// TIA Portal V21 export
FUNCTION_BLOCK "FB603"   // FB603, LAD
TITLE = FB603
{ S7_Optimized_Access := 'FALSE' }
AUTHOR : PRECISE
FAMILY : PRECISE
// CIP
// stored: AutoNumber false, SetENOAutomatically false
   VAR_INPUT
      CycleEnable : Bool;
      CycleRunning : Bool;
      SecPulse : Bool;
      AlwaysTrue : Bool;
      CycleSelection : "CIP";
      ConductivitySuccessWhileRinse : Bool;
      ConductivitySuccessWhileDrain : Bool;
      ConductivitySuccessWhileTransfer : Bool;
   END_VAR
   VAR_OUTPUT
      Started : Bool;
      VentValve : Bool;
      PrintActualRep : Int;
   END_VAR
   VAR_IN_OUT
      Over : Bool;
      OverTemp : Bool;
      RepeatCycle : Bool;
      ActualRepetition : Int;
      CycleStart : "CipCycleStarted";
      CycleOver : "CipCycleOver";
      ConductivityStatus : Bool;
      TimeSaveModeRep : Int;
      StartFillingToSaveTime : Bool;
      Reset : Bool;
      RecirculationPopupTemp : Bool;
      RecirculationPopupTempAck : Bool;
   END_VAR
   VAR
      Re : Array[0..30] of Bool;
   END_VAR
   VAR_TEMP   // added for the SCL form of the ladder/FBD networks
      _w1 : Bool;
      _w2 : Bool;
      _w3 : Bool;
      _w4 : Bool;
      _w5 : Bool;
      _w6 : Bool;
      _w7 : Bool;
      _w8 : Bool;
      _w9 : Bool;
      _w10 : Bool;
      _w11 : Bool;
      _w12 : Bool;
   END_VAR
BEGIN

REGION Network 1
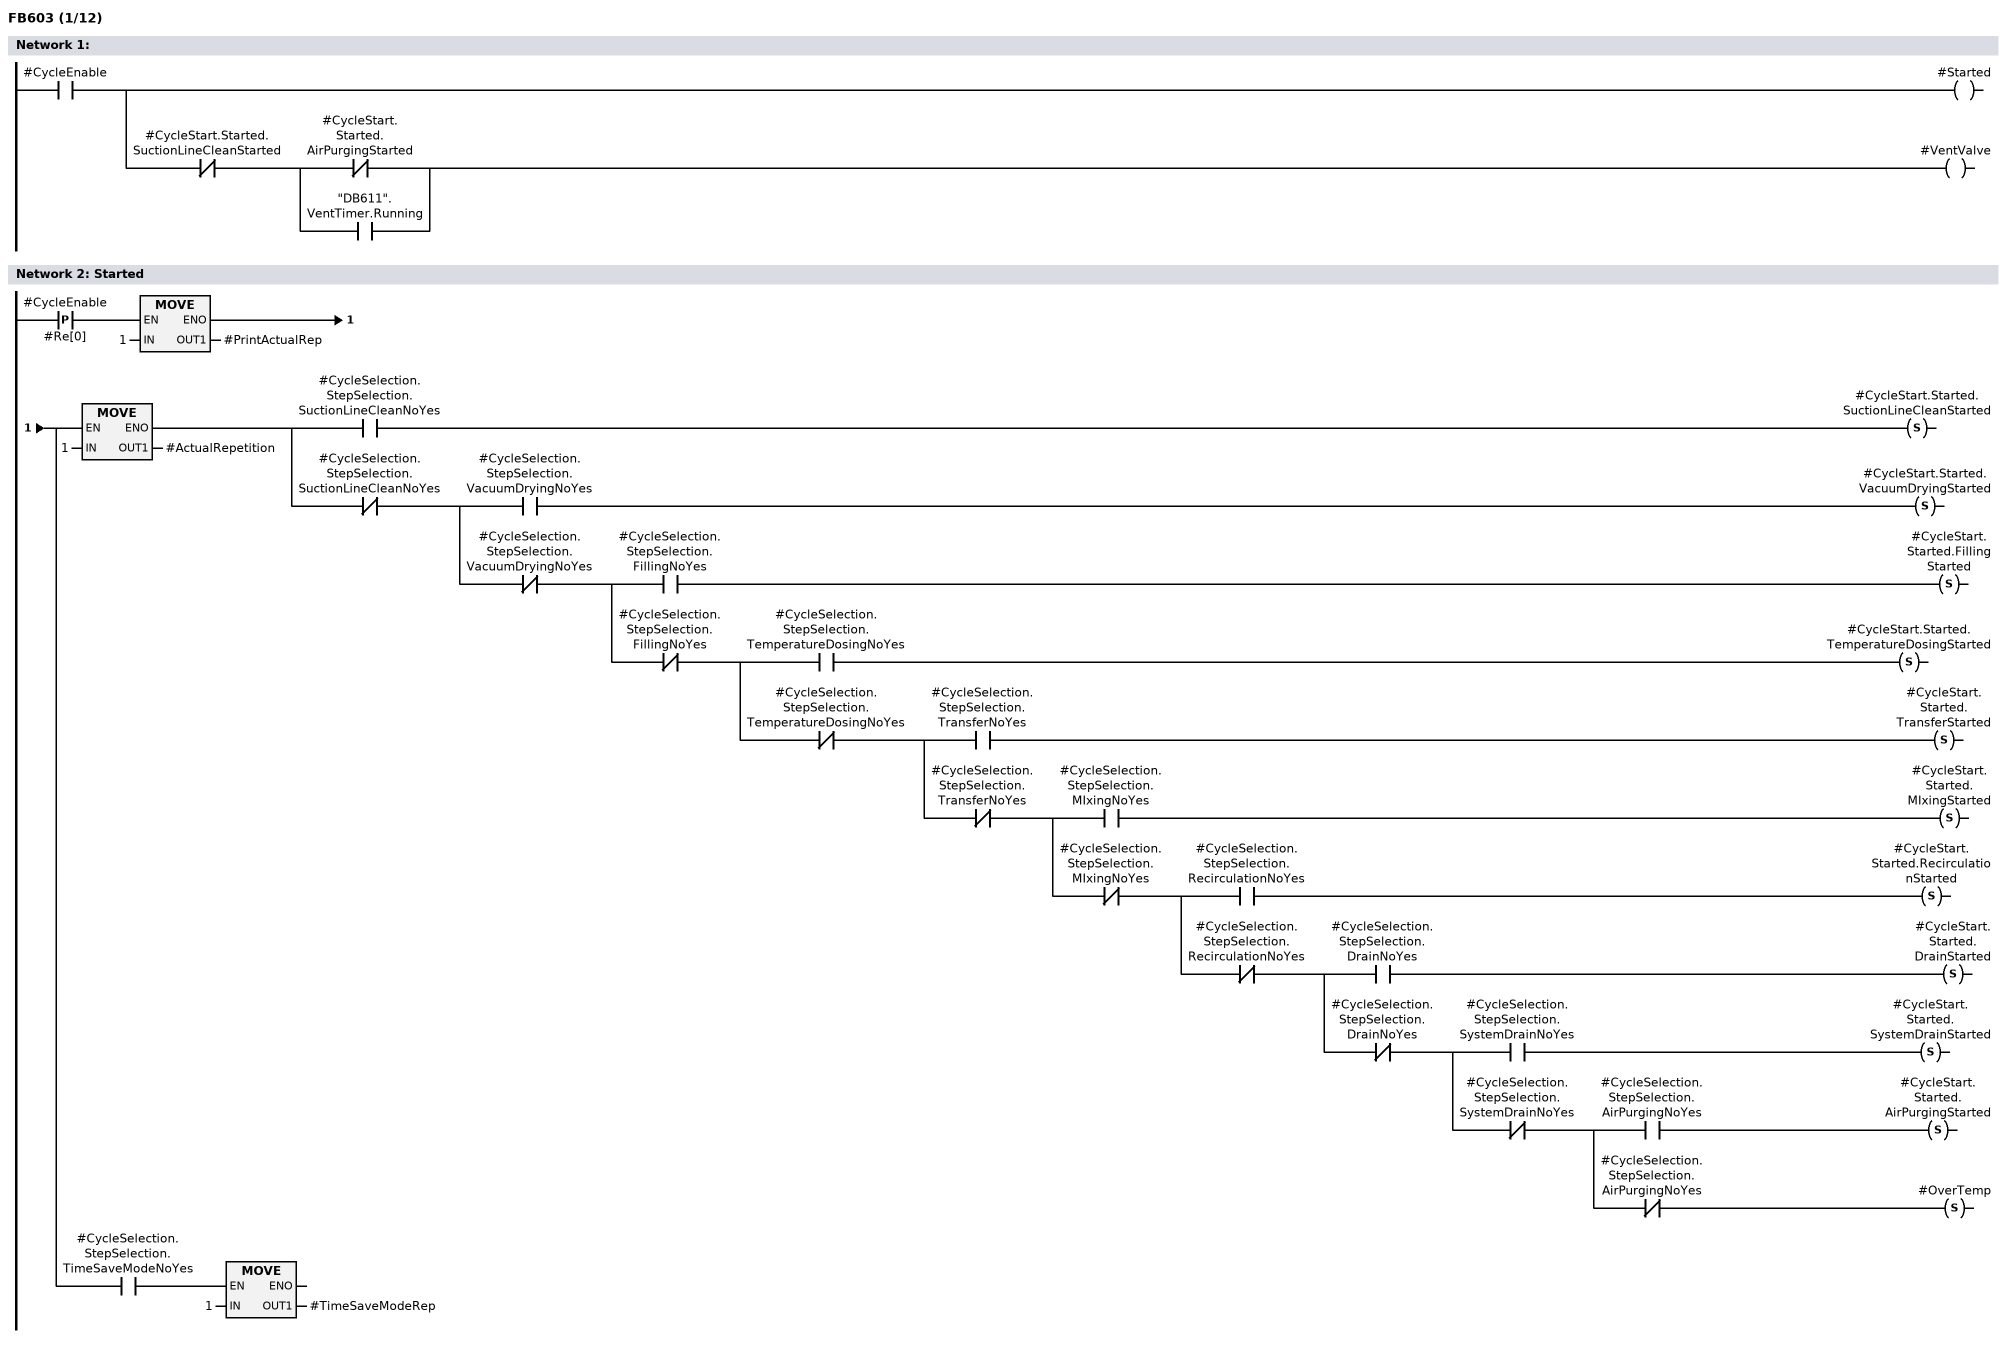
   RUNG wire#powerrail
      Contact( #CycleEnable )
      wire#w1
      Coil( #Started )
   END_RUNG
   RUNG wire#w1
      I_Contact( #CycleStart.Started.SuctionLineCleanStarted )
      wire#w2
      I_Contact( #CycleStart.Started.AirPurgingStarted )
      wire#w3
      Coil( #VentValve )
   END_RUNG
   RUNG wire#w2
      Contact( "DB611".VentTimer.Running )
   END_RUNG wire#w3
   // the same network as SCL:
   #Started := #CycleEnable;
   #VentValve := #CycleEnable AND NOT #CycleStart.Started.SuctionLineCleanStarted AND (NOT #CycleStart.Started.AirPurgingStarted OR "DB611".VentTimer.Running);
END_REGION

REGION Network 2: Started
   RUNG wire#powerrail
      P_Contact(operand := #CycleEnable, bit := #Re[0])
      Move(in := 1, out1 => #PrintActualRep)
      wire#w1
      Move(in := 1, out1 => #ActualRepetition)
      wire#w2
      Contact( #CycleSelection.StepSelection.SuctionLineCleanNoYes )
      S_Coil( #CycleStart.Started.SuctionLineCleanStarted )
   END_RUNG
   RUNG wire#w2
      I_Contact( #CycleSelection.StepSelection.SuctionLineCleanNoYes )
      wire#w3
      Contact( #CycleSelection.StepSelection.VacuumDryingNoYes )
      S_Coil( #CycleStart.Started.VacuumDryingStarted )
   END_RUNG
   RUNG wire#w3
      I_Contact( #CycleSelection.StepSelection.VacuumDryingNoYes )
      wire#w4
      Contact( #CycleSelection.StepSelection.FillingNoYes )
      S_Coil( #CycleStart.Started.FillingStarted )
   END_RUNG
   RUNG wire#w4
      I_Contact( #CycleSelection.StepSelection.FillingNoYes )
      wire#w5
      Contact( #CycleSelection.StepSelection.TemperatureDosingNoYes )
      S_Coil( #CycleStart.Started.TemperatureDosingStarted )
   END_RUNG
   RUNG wire#w5
      I_Contact( #CycleSelection.StepSelection.TemperatureDosingNoYes )
      wire#w6
      Contact( #CycleSelection.StepSelection.TransferNoYes )
      S_Coil( #CycleStart.Started.TransferStarted )
   END_RUNG
   RUNG wire#w6
      I_Contact( #CycleSelection.StepSelection.TransferNoYes )
      wire#w7
      Contact( #CycleSelection.StepSelection.MIxingNoYes )
      S_Coil( #CycleStart.Started.MIxingStarted )
   END_RUNG
   RUNG wire#w7
      I_Contact( #CycleSelection.StepSelection.MIxingNoYes )
      wire#w8
      Contact( #CycleSelection.StepSelection.RecirculationNoYes )
      S_Coil( #CycleStart.Started.RecirculationStarted )
   END_RUNG
   RUNG wire#w8
      I_Contact( #CycleSelection.StepSelection.RecirculationNoYes )
      wire#w9
      Contact( #CycleSelection.StepSelection.DrainNoYes )
      S_Coil( #CycleStart.Started.DrainStarted )
   END_RUNG
   RUNG wire#w9
      I_Contact( #CycleSelection.StepSelection.DrainNoYes )
      wire#w10
      Contact( #CycleSelection.StepSelection.SystemDrainNoYes )
      S_Coil( #CycleStart.Started.SystemDrainStarted )
   END_RUNG
   RUNG wire#w10
      I_Contact( #CycleSelection.StepSelection.SystemDrainNoYes )
      wire#w11
      Contact( #CycleSelection.StepSelection.AirPurgingNoYes )
      S_Coil( #CycleStart.Started.AirPurgingStarted )
   END_RUNG
   RUNG wire#w11
      I_Contact( #CycleSelection.StepSelection.AirPurgingNoYes )
      S_Coil( #OverTemp )
   END_RUNG
   RUNG wire#w1
      Contact( #CycleSelection.StepSelection.TimeSaveModeNoYes )
      Move(in := 1, out1 => #TimeSaveModeRep)
   END_RUNG
   // the same network as SCL:
   #_w1 := #CycleEnable AND NOT #Re[0];   // rising edge of #CycleEnable
   #Re[0] := #CycleEnable;
   IF #_w1 THEN
       #PrintActualRep := 1;
       #ActualRepetition := 1;
   END_IF;
   IF #_w1 AND #CycleSelection.StepSelection.SuctionLineCleanNoYes THEN
       #CycleStart.Started.SuctionLineCleanStarted := TRUE;
   END_IF;
   #_w2 := #_w1 AND NOT #CycleSelection.StepSelection.SuctionLineCleanNoYes;
   IF #_w2 AND #CycleSelection.StepSelection.VacuumDryingNoYes THEN
       #CycleStart.Started.VacuumDryingStarted := TRUE;
   END_IF;
   #_w3 := #_w2 AND NOT #CycleSelection.StepSelection.VacuumDryingNoYes;
   IF #_w3 AND #CycleSelection.StepSelection.FillingNoYes THEN
       #CycleStart.Started.FillingStarted := TRUE;
   END_IF;
   #_w4 := #_w3 AND NOT #CycleSelection.StepSelection.FillingNoYes;
   IF #_w4 AND #CycleSelection.StepSelection.TemperatureDosingNoYes THEN
       #CycleStart.Started.TemperatureDosingStarted := TRUE;
   END_IF;
   #_w5 := #_w4 AND NOT #CycleSelection.StepSelection.TemperatureDosingNoYes;
   IF #_w5 AND #CycleSelection.StepSelection.TransferNoYes THEN
       #CycleStart.Started.TransferStarted := TRUE;
   END_IF;
   #_w6 := #_w5 AND NOT #CycleSelection.StepSelection.TransferNoYes;
   IF #_w6 AND #CycleSelection.StepSelection.MIxingNoYes THEN
       #CycleStart.Started.MIxingStarted := TRUE;
   END_IF;
   #_w7 := #_w6 AND NOT #CycleSelection.StepSelection.MIxingNoYes;
   IF #_w7 AND #CycleSelection.StepSelection.RecirculationNoYes THEN
       #CycleStart.Started.RecirculationStarted := TRUE;
   END_IF;
   #_w8 := #_w7 AND NOT #CycleSelection.StepSelection.RecirculationNoYes;
   IF #_w8 AND #CycleSelection.StepSelection.DrainNoYes THEN
       #CycleStart.Started.DrainStarted := TRUE;
   END_IF;
   #_w9 := #_w8 AND NOT #CycleSelection.StepSelection.DrainNoYes;
   IF #_w9 AND #CycleSelection.StepSelection.SystemDrainNoYes THEN
       #CycleStart.Started.SystemDrainStarted := TRUE;
   END_IF;
   #_w10 := #_w9 AND NOT #CycleSelection.StepSelection.SystemDrainNoYes;
   IF #_w10 AND #CycleSelection.StepSelection.AirPurgingNoYes THEN
       #CycleStart.Started.AirPurgingStarted := TRUE;
   END_IF;
   IF #_w10 AND NOT #CycleSelection.StepSelection.AirPurgingNoYes THEN #OverTemp := TRUE; END_IF;
   IF #_w1 AND #CycleSelection.StepSelection.TimeSaveModeNoYes THEN #TimeSaveModeRep := 1; END_IF;
END_REGION

REGION Network 3: SuctionLineCleanOver
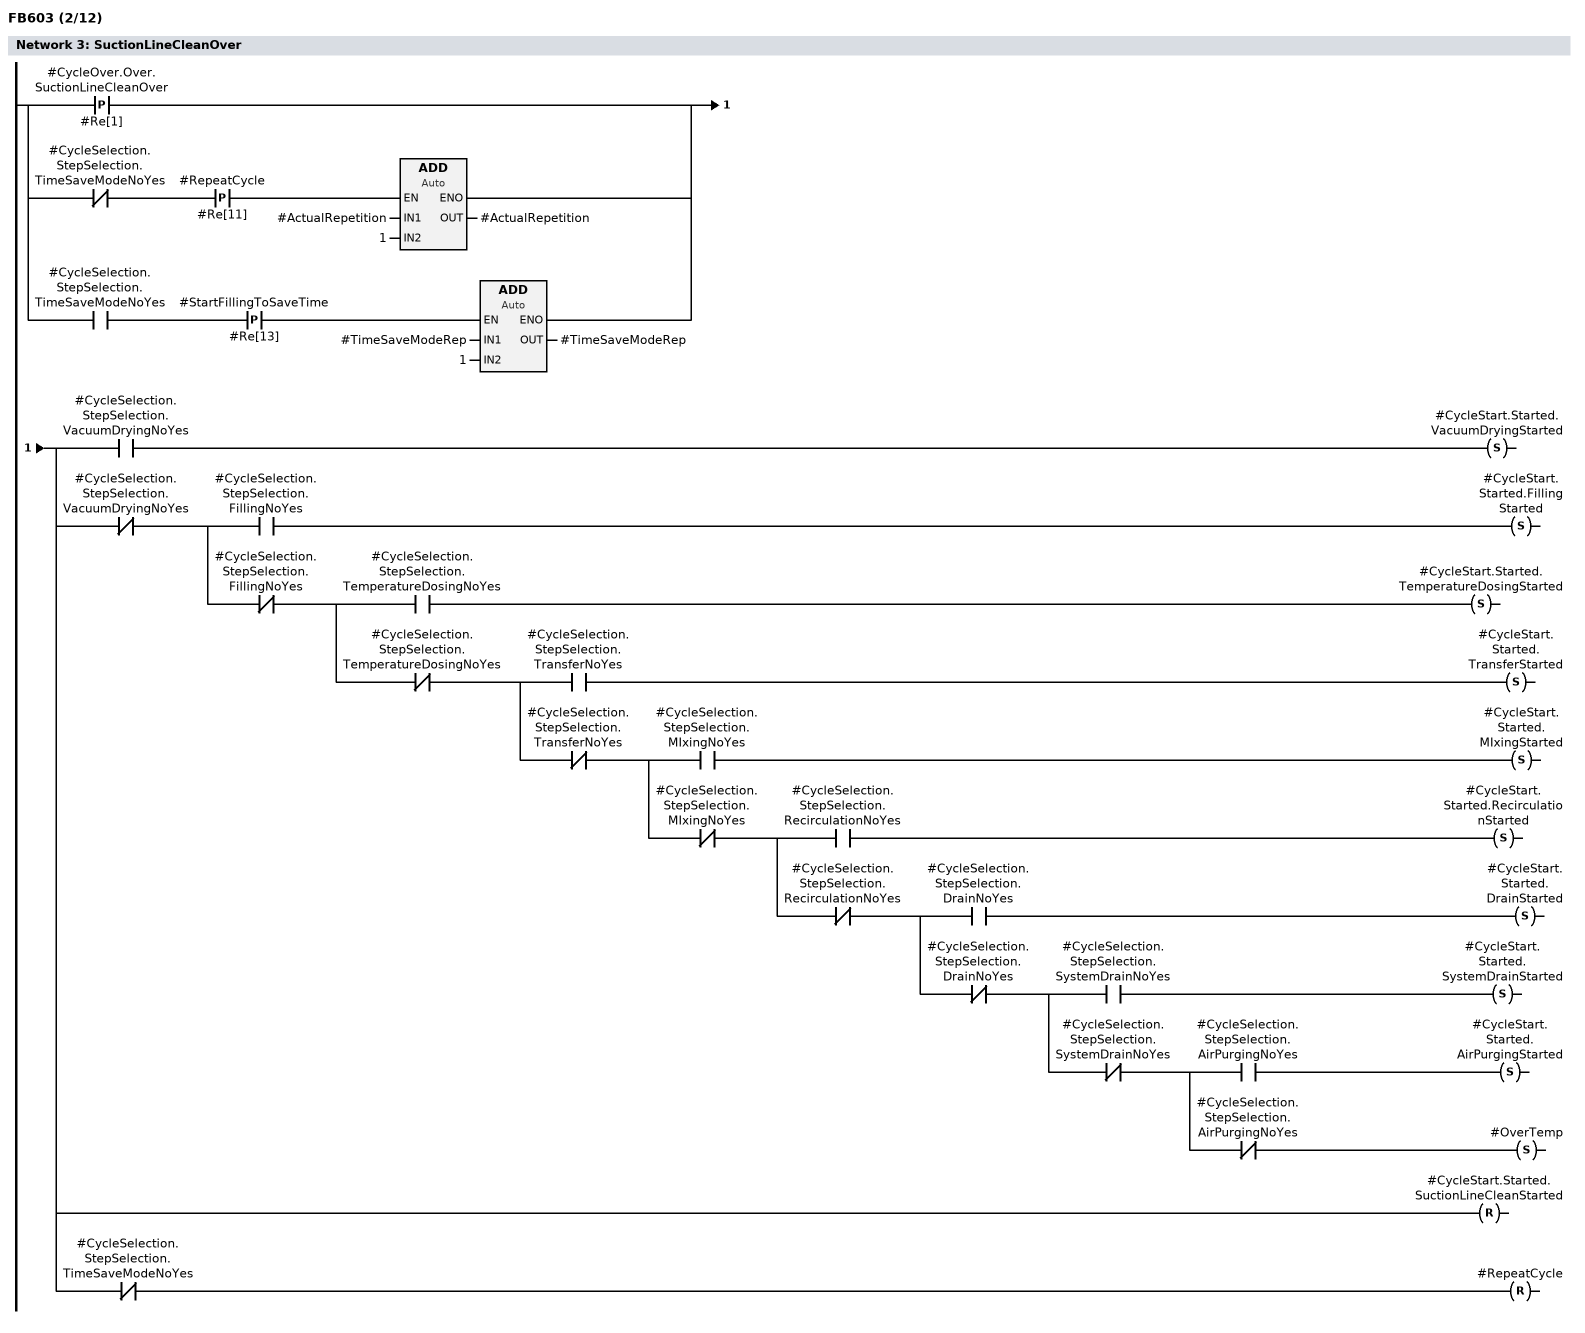
   RUNG wire#powerrail
      P_Contact(operand := #CycleOver.Over.SuctionLineCleanOver, bit := #Re[1])
      wire#w1
      Contact( #CycleSelection.StepSelection.VacuumDryingNoYes )
      S_Coil( #CycleStart.Started.VacuumDryingStarted )
   END_RUNG
   RUNG wire#powerrail
      I_Contact( #CycleSelection.StepSelection.TimeSaveModeNoYes )
      P_Contact(operand := #RepeatCycle, bit := #Re[11])
      Add(in1 := #ActualRepetition, in2 := 1, out => #ActualRepetition)
   END_RUNG wire#w1
   RUNG wire#powerrail
      Contact( #CycleSelection.StepSelection.TimeSaveModeNoYes )
      P_Contact(operand := #StartFillingToSaveTime, bit := #Re[13])
      Add(in1 := #TimeSaveModeRep, in2 := 1, out => #TimeSaveModeRep)
   END_RUNG wire#w1
   RUNG wire#w1
      I_Contact( #CycleSelection.StepSelection.VacuumDryingNoYes )
      wire#w2
      Contact( #CycleSelection.StepSelection.FillingNoYes )
      S_Coil( #CycleStart.Started.FillingStarted )
   END_RUNG
   RUNG wire#w2
      I_Contact( #CycleSelection.StepSelection.FillingNoYes )
      wire#w3
      Contact( #CycleSelection.StepSelection.TemperatureDosingNoYes )
      S_Coil( #CycleStart.Started.TemperatureDosingStarted )
   END_RUNG
   RUNG wire#w3
      I_Contact( #CycleSelection.StepSelection.TemperatureDosingNoYes )
      wire#w4
      Contact( #CycleSelection.StepSelection.TransferNoYes )
      S_Coil( #CycleStart.Started.TransferStarted )
   END_RUNG
   RUNG wire#w4
      I_Contact( #CycleSelection.StepSelection.TransferNoYes )
      wire#w5
      Contact( #CycleSelection.StepSelection.MIxingNoYes )
      S_Coil( #CycleStart.Started.MIxingStarted )
   END_RUNG
   RUNG wire#w5
      I_Contact( #CycleSelection.StepSelection.MIxingNoYes )
      wire#w6
      Contact( #CycleSelection.StepSelection.RecirculationNoYes )
      S_Coil( #CycleStart.Started.RecirculationStarted )
   END_RUNG
   RUNG wire#w6
      I_Contact( #CycleSelection.StepSelection.RecirculationNoYes )
      wire#w7
      Contact( #CycleSelection.StepSelection.DrainNoYes )
      S_Coil( #CycleStart.Started.DrainStarted )
   END_RUNG
   RUNG wire#w7
      I_Contact( #CycleSelection.StepSelection.DrainNoYes )
      wire#w8
      Contact( #CycleSelection.StepSelection.SystemDrainNoYes )
      S_Coil( #CycleStart.Started.SystemDrainStarted )
   END_RUNG
   RUNG wire#w8
      I_Contact( #CycleSelection.StepSelection.SystemDrainNoYes )
      wire#w9
      Contact( #CycleSelection.StepSelection.AirPurgingNoYes )
      S_Coil( #CycleStart.Started.AirPurgingStarted )
   END_RUNG
   RUNG wire#w9
      I_Contact( #CycleSelection.StepSelection.AirPurgingNoYes )
      S_Coil( #OverTemp )
   END_RUNG
   RUNG wire#w1
      R_Coil( #CycleStart.Started.SuctionLineCleanStarted )
   END_RUNG
   RUNG wire#w1
      I_Contact( #CycleSelection.StepSelection.TimeSaveModeNoYes )
      R_Coil( #RepeatCycle )
   END_RUNG
   // the same network as SCL:
   #_w1 := #CycleOver.Over.SuctionLineCleanOver AND NOT #Re[1];   // rising edge of #CycleOver.Over.SuctionLineCleanOver
   #Re[1] := #CycleOver.Over.SuctionLineCleanOver;
   #_w2 := NOT #CycleSelection.StepSelection.TimeSaveModeNoYes AND #RepeatCycle AND NOT #Re[11];   // rising edge of #RepeatCycle
   #Re[11] := #RepeatCycle;
   IF #_w2 THEN #ActualRepetition := #ActualRepetition + 1; END_IF;
   #_w3 := #CycleSelection.StepSelection.TimeSaveModeNoYes AND #StartFillingToSaveTime AND NOT #Re[13];   // rising edge of #StartFillingToSaveTime
   #Re[13] := #StartFillingToSaveTime;
   IF #_w3 THEN #TimeSaveModeRep := #TimeSaveModeRep + 1; END_IF;
   #_w4 := #_w1 OR #_w2 OR #_w3;
   IF #_w4 AND #CycleSelection.StepSelection.VacuumDryingNoYes THEN
       #CycleStart.Started.VacuumDryingStarted := TRUE;
   END_IF;
   #_w5 := #_w4 AND NOT #CycleSelection.StepSelection.VacuumDryingNoYes;
   IF #_w5 AND #CycleSelection.StepSelection.FillingNoYes THEN
       #CycleStart.Started.FillingStarted := TRUE;
   END_IF;
   #_w6 := #_w5 AND NOT #CycleSelection.StepSelection.FillingNoYes;
   IF #_w6 AND #CycleSelection.StepSelection.TemperatureDosingNoYes THEN
       #CycleStart.Started.TemperatureDosingStarted := TRUE;
   END_IF;
   #_w7 := #_w6 AND NOT #CycleSelection.StepSelection.TemperatureDosingNoYes;
   IF #_w7 AND #CycleSelection.StepSelection.TransferNoYes THEN
       #CycleStart.Started.TransferStarted := TRUE;
   END_IF;
   #_w8 := #_w7 AND NOT #CycleSelection.StepSelection.TransferNoYes;
   IF #_w8 AND #CycleSelection.StepSelection.MIxingNoYes THEN
       #CycleStart.Started.MIxingStarted := TRUE;
   END_IF;
   #_w9 := #_w8 AND NOT #CycleSelection.StepSelection.MIxingNoYes;
   IF #_w9 AND #CycleSelection.StepSelection.RecirculationNoYes THEN
       #CycleStart.Started.RecirculationStarted := TRUE;
   END_IF;
   #_w10 := #_w9 AND NOT #CycleSelection.StepSelection.RecirculationNoYes;
   IF #_w10 AND #CycleSelection.StepSelection.DrainNoYes THEN
       #CycleStart.Started.DrainStarted := TRUE;
   END_IF;
   #_w11 := #_w10 AND NOT #CycleSelection.StepSelection.DrainNoYes;
   IF #_w11 AND #CycleSelection.StepSelection.SystemDrainNoYes THEN
       #CycleStart.Started.SystemDrainStarted := TRUE;
   END_IF;
   #_w12 := #_w11 AND NOT #CycleSelection.StepSelection.SystemDrainNoYes;
   IF #_w12 AND #CycleSelection.StepSelection.AirPurgingNoYes THEN
       #CycleStart.Started.AirPurgingStarted := TRUE;
   END_IF;
   IF #_w12 AND NOT #CycleSelection.StepSelection.AirPurgingNoYes THEN #OverTemp := TRUE; END_IF;
   IF #_w4 THEN #CycleStart.Started.SuctionLineCleanStarted := FALSE; END_IF;
   IF #_w4 AND NOT #CycleSelection.StepSelection.TimeSaveModeNoYes THEN #RepeatCycle := FALSE; END_IF;
END_REGION

REGION Network 4: VacuumDryingOver
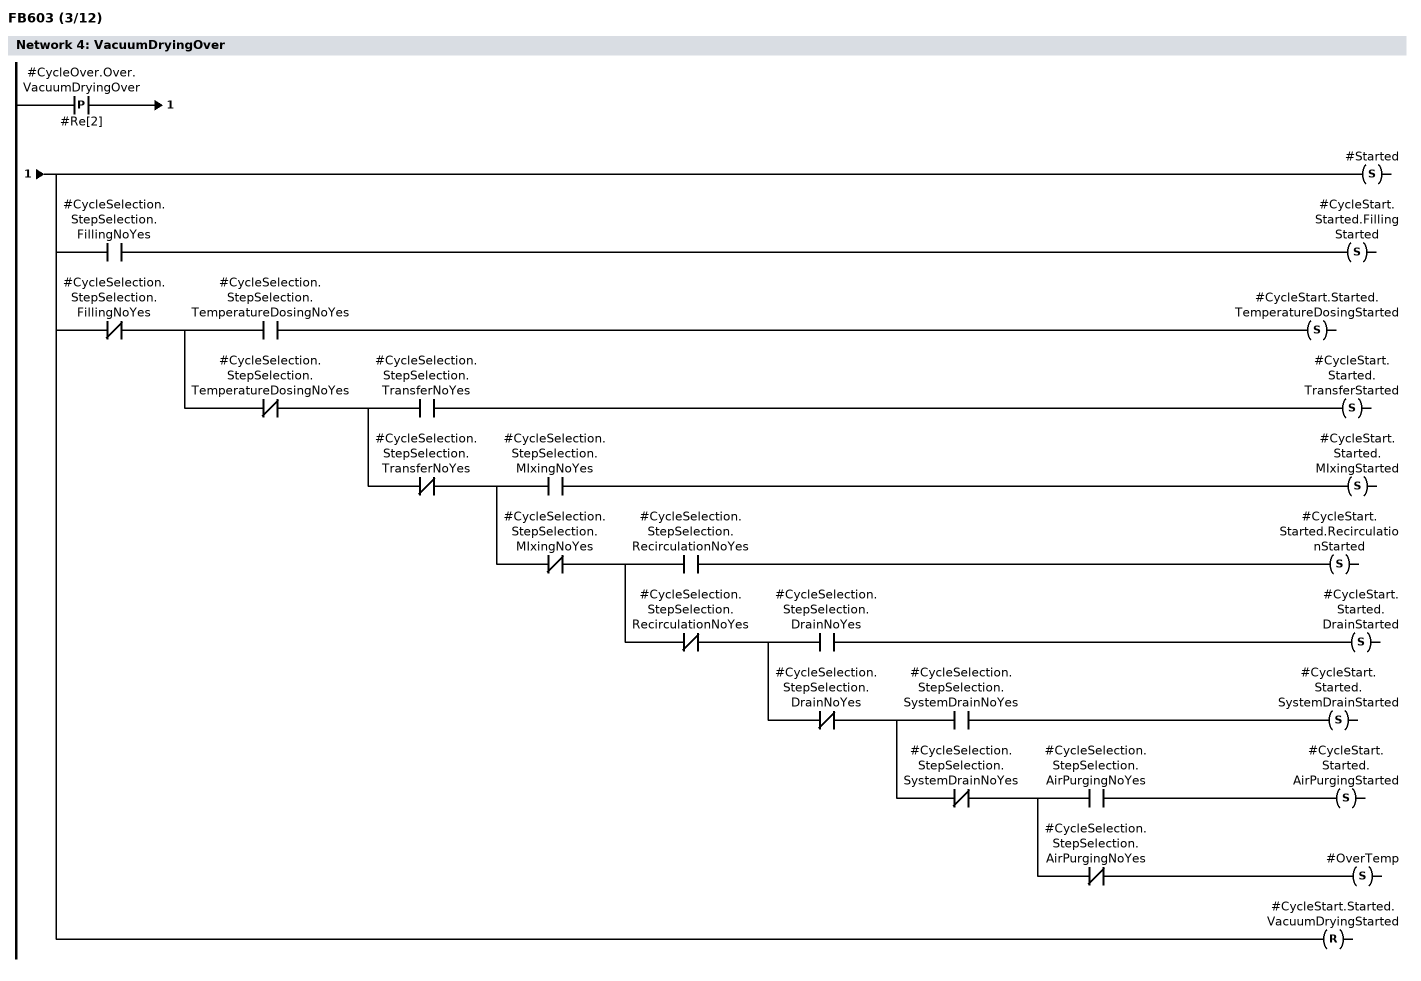
   RUNG wire#powerrail
      P_Contact(operand := #CycleOver.Over.VacuumDryingOver, bit := #Re[2])
      wire#w1
      S_Coil( #Started )
   END_RUNG
   RUNG wire#w1
      Contact( #CycleSelection.StepSelection.FillingNoYes )
      S_Coil( #CycleStart.Started.FillingStarted )
   END_RUNG
   RUNG wire#w1
      I_Contact( #CycleSelection.StepSelection.FillingNoYes )
      wire#w2
      Contact( #CycleSelection.StepSelection.TemperatureDosingNoYes )
      S_Coil( #CycleStart.Started.TemperatureDosingStarted )
   END_RUNG
   RUNG wire#w2
      I_Contact( #CycleSelection.StepSelection.TemperatureDosingNoYes )
      wire#w3
      Contact( #CycleSelection.StepSelection.TransferNoYes )
      S_Coil( #CycleStart.Started.TransferStarted )
   END_RUNG
   RUNG wire#w3
      I_Contact( #CycleSelection.StepSelection.TransferNoYes )
      wire#w4
      Contact( #CycleSelection.StepSelection.MIxingNoYes )
      S_Coil( #CycleStart.Started.MIxingStarted )
   END_RUNG
   RUNG wire#w4
      I_Contact( #CycleSelection.StepSelection.MIxingNoYes )
      wire#w5
      Contact( #CycleSelection.StepSelection.RecirculationNoYes )
      S_Coil( #CycleStart.Started.RecirculationStarted )
   END_RUNG
   RUNG wire#w5
      I_Contact( #CycleSelection.StepSelection.RecirculationNoYes )
      wire#w6
      Contact( #CycleSelection.StepSelection.DrainNoYes )
      S_Coil( #CycleStart.Started.DrainStarted )
   END_RUNG
   RUNG wire#w6
      I_Contact( #CycleSelection.StepSelection.DrainNoYes )
      wire#w7
      Contact( #CycleSelection.StepSelection.SystemDrainNoYes )
      S_Coil( #CycleStart.Started.SystemDrainStarted )
   END_RUNG
   RUNG wire#w7
      I_Contact( #CycleSelection.StepSelection.SystemDrainNoYes )
      wire#w8
      Contact( #CycleSelection.StepSelection.AirPurgingNoYes )
      S_Coil( #CycleStart.Started.AirPurgingStarted )
   END_RUNG
   RUNG wire#w8
      I_Contact( #CycleSelection.StepSelection.AirPurgingNoYes )
      S_Coil( #OverTemp )
   END_RUNG
   RUNG wire#w1
      R_Coil( #CycleStart.Started.VacuumDryingStarted )
   END_RUNG
   // the same network as SCL:
   #_w1 := #CycleOver.Over.VacuumDryingOver AND NOT #Re[2];   // rising edge of #CycleOver.Over.VacuumDryingOver
   #Re[2] := #CycleOver.Over.VacuumDryingOver;
   IF #_w1 THEN #Started := TRUE; END_IF;
   IF #_w1 AND #CycleSelection.StepSelection.FillingNoYes THEN
       #CycleStart.Started.FillingStarted := TRUE;
   END_IF;
   #_w2 := #_w1 AND NOT #CycleSelection.StepSelection.FillingNoYes;
   IF #_w2 AND #CycleSelection.StepSelection.TemperatureDosingNoYes THEN
       #CycleStart.Started.TemperatureDosingStarted := TRUE;
   END_IF;
   #_w3 := #_w2 AND NOT #CycleSelection.StepSelection.TemperatureDosingNoYes;
   IF #_w3 AND #CycleSelection.StepSelection.TransferNoYes THEN
       #CycleStart.Started.TransferStarted := TRUE;
   END_IF;
   #_w4 := #_w3 AND NOT #CycleSelection.StepSelection.TransferNoYes;
   IF #_w4 AND #CycleSelection.StepSelection.MIxingNoYes THEN
       #CycleStart.Started.MIxingStarted := TRUE;
   END_IF;
   #_w5 := #_w4 AND NOT #CycleSelection.StepSelection.MIxingNoYes;
   IF #_w5 AND #CycleSelection.StepSelection.RecirculationNoYes THEN
       #CycleStart.Started.RecirculationStarted := TRUE;
   END_IF;
   #_w6 := #_w5 AND NOT #CycleSelection.StepSelection.RecirculationNoYes;
   IF #_w6 AND #CycleSelection.StepSelection.DrainNoYes THEN
       #CycleStart.Started.DrainStarted := TRUE;
   END_IF;
   #_w7 := #_w6 AND NOT #CycleSelection.StepSelection.DrainNoYes;
   IF #_w7 AND #CycleSelection.StepSelection.SystemDrainNoYes THEN
       #CycleStart.Started.SystemDrainStarted := TRUE;
   END_IF;
   #_w8 := #_w7 AND NOT #CycleSelection.StepSelection.SystemDrainNoYes;
   IF #_w8 AND #CycleSelection.StepSelection.AirPurgingNoYes THEN
       #CycleStart.Started.AirPurgingStarted := TRUE;
   END_IF;
   IF #_w8 AND NOT #CycleSelection.StepSelection.AirPurgingNoYes THEN #OverTemp := TRUE; END_IF;
   IF #_w1 THEN #CycleStart.Started.VacuumDryingStarted := FALSE; END_IF;
END_REGION

REGION Network 5: FillOver
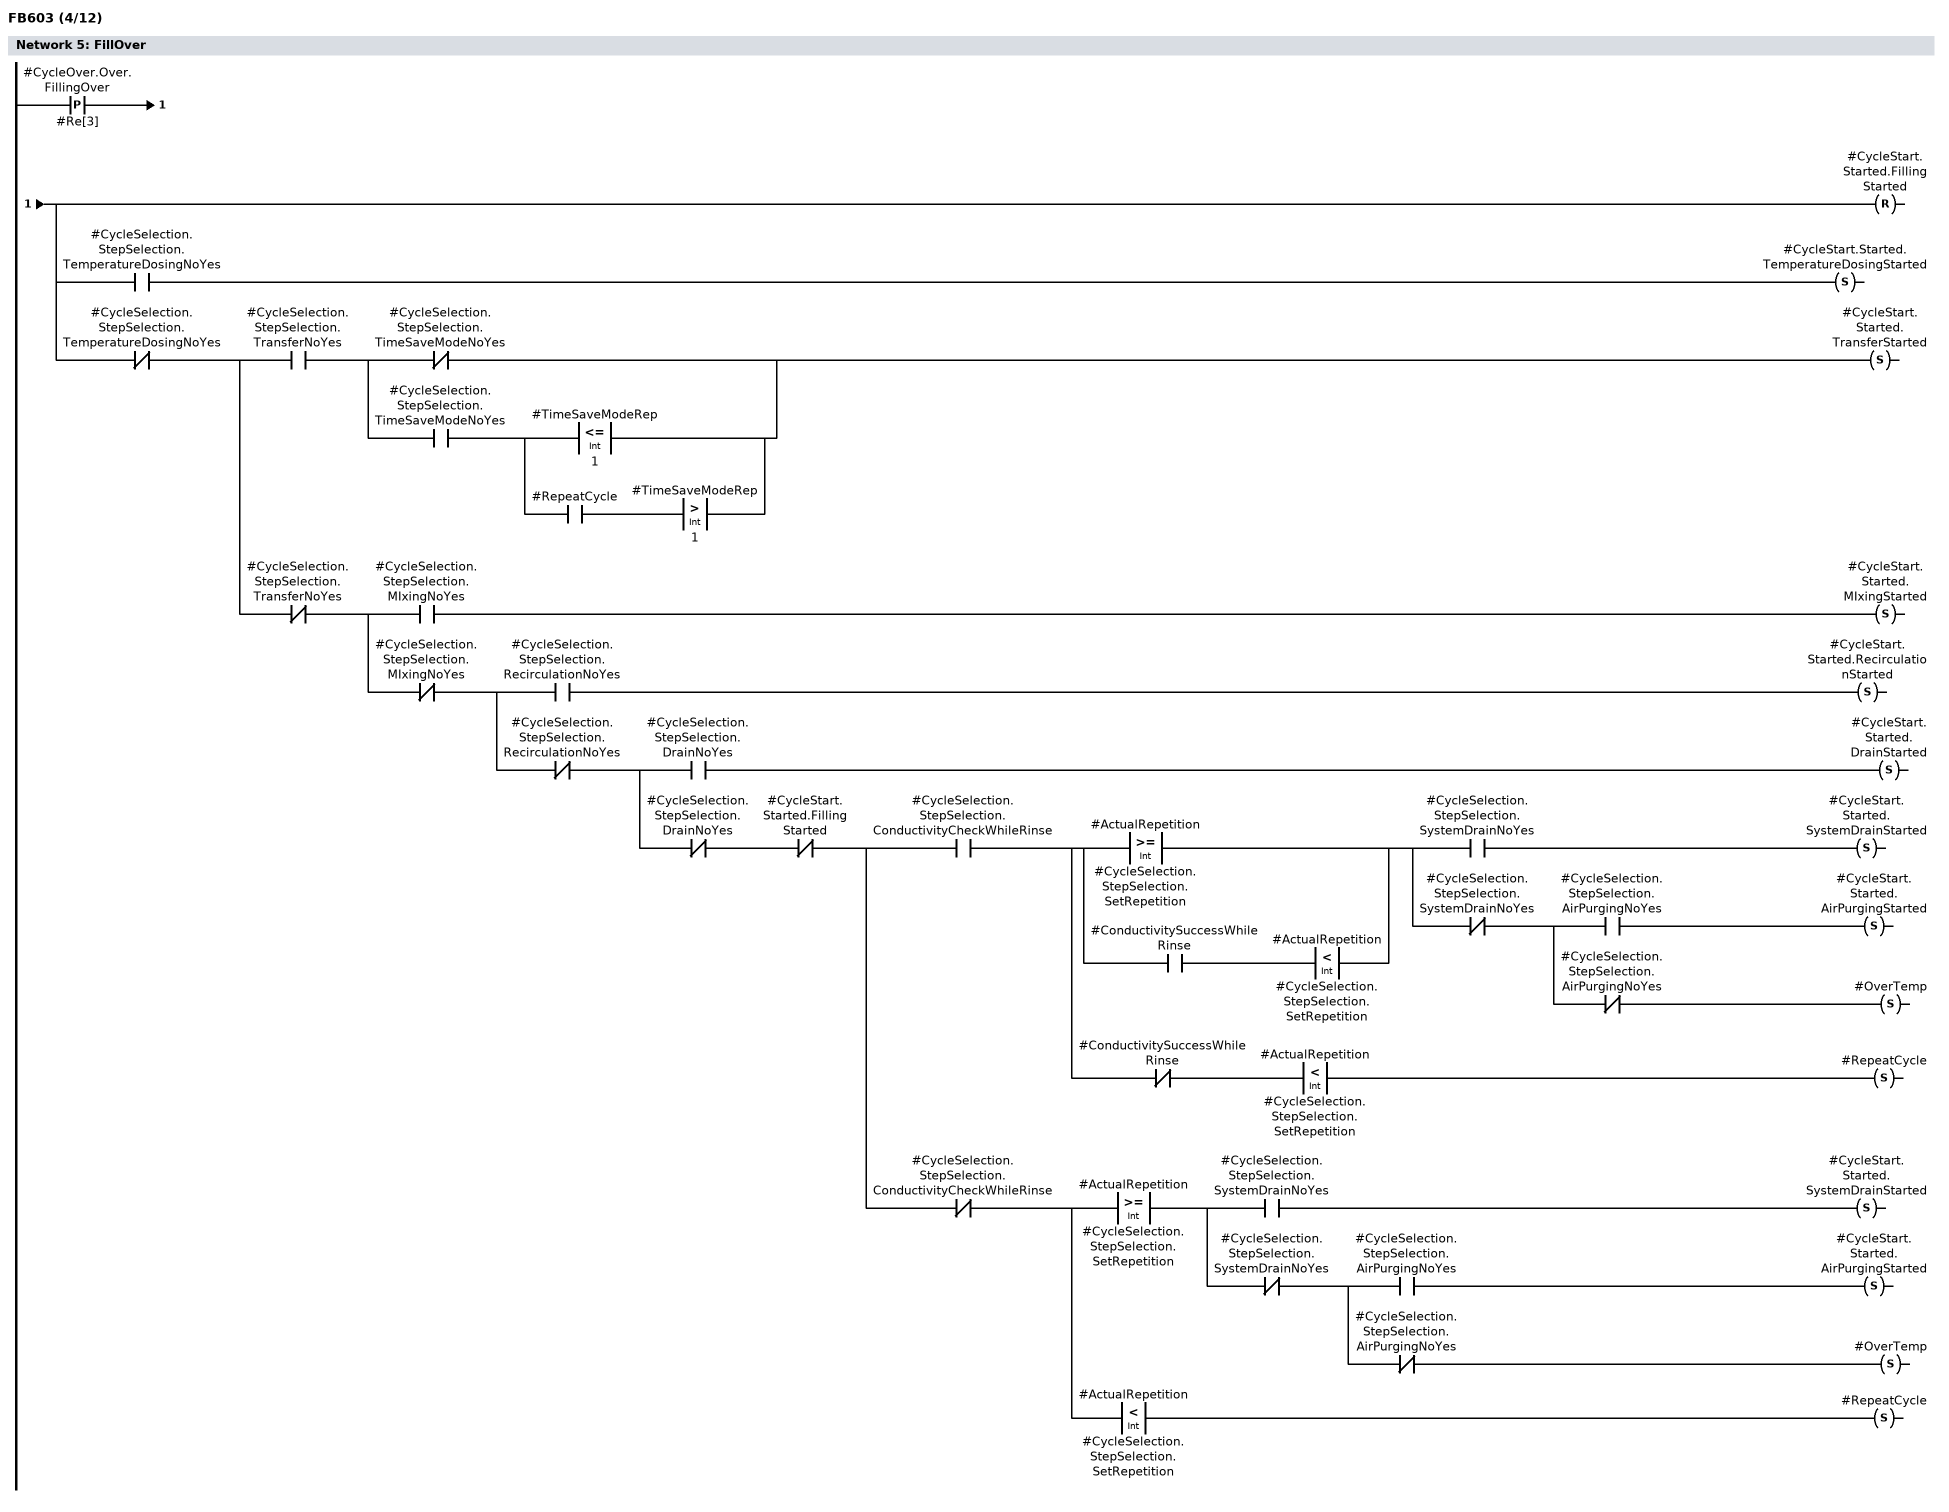
   RUNG wire#powerrail
      P_Contact(operand := #CycleOver.Over.FillingOver, bit := #Re[3])
      wire#w1
      R_Coil( #CycleStart.Started.FillingStarted )
   END_RUNG
   RUNG wire#w1
      Contact( #CycleSelection.StepSelection.TemperatureDosingNoYes )
      S_Coil( #CycleStart.Started.TemperatureDosingStarted )
   END_RUNG
   RUNG wire#w1
      I_Contact( #CycleSelection.StepSelection.TemperatureDosingNoYes )
      wire#w2
      Contact( #CycleSelection.StepSelection.TransferNoYes )
      wire#w3
      I_Contact( #CycleSelection.StepSelection.TimeSaveModeNoYes )
      wire#w4
      S_Coil( #CycleStart.Started.TransferStarted )
   END_RUNG
   RUNG wire#w3
      Contact( #CycleSelection.StepSelection.TimeSaveModeNoYes )
      wire#w5
      { S7_Templates := "SrcType := Int" } LE_Contact(in1 := #TimeSaveModeRep, in2 := 1)
   END_RUNG wire#w4
   RUNG wire#w5
      Contact( #RepeatCycle )
      { S7_Templates := "SrcType := Int" } GT_Contact(in1 := #TimeSaveModeRep, in2 := 1)
   END_RUNG wire#w4
   RUNG wire#w2
      I_Contact( #CycleSelection.StepSelection.TransferNoYes )
      wire#w6
      Contact( #CycleSelection.StepSelection.MIxingNoYes )
      S_Coil( #CycleStart.Started.MIxingStarted )
   END_RUNG
   RUNG wire#w6
      I_Contact( #CycleSelection.StepSelection.MIxingNoYes )
      wire#w7
      Contact( #CycleSelection.StepSelection.RecirculationNoYes )
      S_Coil( #CycleStart.Started.RecirculationStarted )
   END_RUNG
   RUNG wire#w7
      I_Contact( #CycleSelection.StepSelection.RecirculationNoYes )
      wire#w8
      Contact( #CycleSelection.StepSelection.DrainNoYes )
      S_Coil( #CycleStart.Started.DrainStarted )
   END_RUNG
   RUNG wire#w8
      I_Contact( #CycleSelection.StepSelection.DrainNoYes )
      I_Contact( #CycleStart.Started.FillingStarted )
      wire#w9
      Contact( #CycleSelection.StepSelection.ConductivityCheckWhileRinse )
      wire#w10
      { S7_Templates := "SrcType := Int" } GE_Contact(in1 := #ActualRepetition, in2 := #CycleSelection.StepSelection.SetRepetition)
      wire#w11
      Contact( #CycleSelection.StepSelection.SystemDrainNoYes )
      S_Coil( #CycleStart.Started.SystemDrainStarted )
   END_RUNG
   RUNG wire#w10
      Contact( #ConductivitySuccessWhileRinse )
      { S7_Templates := "SrcType := Int" } LT_Contact(in1 := #ActualRepetition, in2 := #CycleSelection.StepSelection.SetRepetition)
   END_RUNG wire#w11
   RUNG wire#w11
      I_Contact( #CycleSelection.StepSelection.SystemDrainNoYes )
      wire#w12
      Contact( #CycleSelection.StepSelection.AirPurgingNoYes )
      S_Coil( #CycleStart.Started.AirPurgingStarted )
   END_RUNG
   RUNG wire#w12
      I_Contact( #CycleSelection.StepSelection.AirPurgingNoYes )
      S_Coil( #OverTemp )
   END_RUNG
   RUNG wire#w10
      I_Contact( #ConductivitySuccessWhileRinse )
      { S7_Templates := "SrcType := Int" } LT_Contact(in1 := #ActualRepetition, in2 := #CycleSelection.StepSelection.SetRepetition)
      S_Coil( #RepeatCycle )
   END_RUNG
   RUNG wire#w9
      I_Contact( #CycleSelection.StepSelection.ConductivityCheckWhileRinse )
      wire#w13
      { S7_Templates := "SrcType := Int" } GE_Contact(in1 := #ActualRepetition, in2 := #CycleSelection.StepSelection.SetRepetition)
      wire#w14
      Contact( #CycleSelection.StepSelection.SystemDrainNoYes )
      S_Coil( #CycleStart.Started.SystemDrainStarted )
   END_RUNG
   RUNG wire#w14
      I_Contact( #CycleSelection.StepSelection.SystemDrainNoYes )
      wire#w15
      Contact( #CycleSelection.StepSelection.AirPurgingNoYes )
      S_Coil( #CycleStart.Started.AirPurgingStarted )
   END_RUNG
   RUNG wire#w15
      I_Contact( #CycleSelection.StepSelection.AirPurgingNoYes )
      S_Coil( #OverTemp )
   END_RUNG
   RUNG wire#w13
      { S7_Templates := "SrcType := Int" } LT_Contact(in1 := #ActualRepetition, in2 := #CycleSelection.StepSelection.SetRepetition)
      S_Coil( #RepeatCycle )
   END_RUNG
   // the same network as SCL:
   #_w1 := #CycleOver.Over.FillingOver AND NOT #Re[3];   // rising edge of #CycleOver.Over.FillingOver
   #Re[3] := #CycleOver.Over.FillingOver;
   IF #_w1 THEN #CycleStart.Started.FillingStarted := FALSE; END_IF;
   IF #_w1 AND #CycleSelection.StepSelection.TemperatureDosingNoYes THEN
       #CycleStart.Started.TemperatureDosingStarted := TRUE;
   END_IF;
   #_w2 := #_w1 AND NOT #CycleSelection.StepSelection.TemperatureDosingNoYes;
   IF #_w2 AND #CycleSelection.StepSelection.TransferNoYes AND (NOT #CycleSelection.StepSelection.TimeSaveModeNoYes OR (#CycleSelection.StepSelection.TimeSaveModeNoYes AND ((#TimeSaveModeRep <= 1) OR (#RepeatCycle AND (#TimeSaveModeRep > 1))))) THEN
       #CycleStart.Started.TransferStarted := TRUE;
   END_IF;
   #_w3 := #_w2 AND NOT #CycleSelection.StepSelection.TransferNoYes;
   IF #_w3 AND #CycleSelection.StepSelection.MIxingNoYes THEN
       #CycleStart.Started.MIxingStarted := TRUE;
   END_IF;
   #_w4 := #_w3 AND NOT #CycleSelection.StepSelection.MIxingNoYes;
   IF #_w4 AND #CycleSelection.StepSelection.RecirculationNoYes THEN
       #CycleStart.Started.RecirculationStarted := TRUE;
   END_IF;
   #_w5 := #_w4 AND NOT #CycleSelection.StepSelection.RecirculationNoYes;
   IF #_w5 AND #CycleSelection.StepSelection.DrainNoYes THEN
       #CycleStart.Started.DrainStarted := TRUE;
   END_IF;
   #_w6 := #_w5 AND NOT #CycleSelection.StepSelection.DrainNoYes AND NOT #CycleStart.Started.FillingStarted;
   #_w7 := #_w6 AND #CycleSelection.StepSelection.ConductivityCheckWhileRinse;
   #_w8 := #_w7 AND ((#ActualRepetition >= #CycleSelection.StepSelection.SetRepetition) OR (#ConductivitySuccessWhileRinse AND (#ActualRepetition < #CycleSelection.StepSelection.SetRepetition)));
   IF #_w8 AND #CycleSelection.StepSelection.SystemDrainNoYes THEN
       #CycleStart.Started.SystemDrainStarted := TRUE;
   END_IF;
   #_w9 := #_w8 AND NOT #CycleSelection.StepSelection.SystemDrainNoYes;
   IF #_w9 AND #CycleSelection.StepSelection.AirPurgingNoYes THEN
       #CycleStart.Started.AirPurgingStarted := TRUE;
   END_IF;
   IF #_w9 AND NOT #CycleSelection.StepSelection.AirPurgingNoYes THEN #OverTemp := TRUE; END_IF;
   IF #_w7 AND NOT #ConductivitySuccessWhileRinse AND (#ActualRepetition < #CycleSelection.StepSelection.SetRepetition) THEN
       #RepeatCycle := TRUE;
   END_IF;
   #_w10 := #_w6 AND NOT #CycleSelection.StepSelection.ConductivityCheckWhileRinse;
   #_w11 := #_w10 AND (#ActualRepetition >= #CycleSelection.StepSelection.SetRepetition);
   IF #_w11 AND #CycleSelection.StepSelection.SystemDrainNoYes THEN
       #CycleStart.Started.SystemDrainStarted := TRUE;
   END_IF;
   #_w12 := #_w11 AND NOT #CycleSelection.StepSelection.SystemDrainNoYes;
   IF #_w12 AND #CycleSelection.StepSelection.AirPurgingNoYes THEN
       #CycleStart.Started.AirPurgingStarted := TRUE;
   END_IF;
   IF #_w12 AND NOT #CycleSelection.StepSelection.AirPurgingNoYes THEN #OverTemp := TRUE; END_IF;
   IF #_w10 AND (#ActualRepetition < #CycleSelection.StepSelection.SetRepetition) THEN
       #RepeatCycle := TRUE;
   END_IF;
END_REGION

REGION Network 6: TemperatureDosingOver
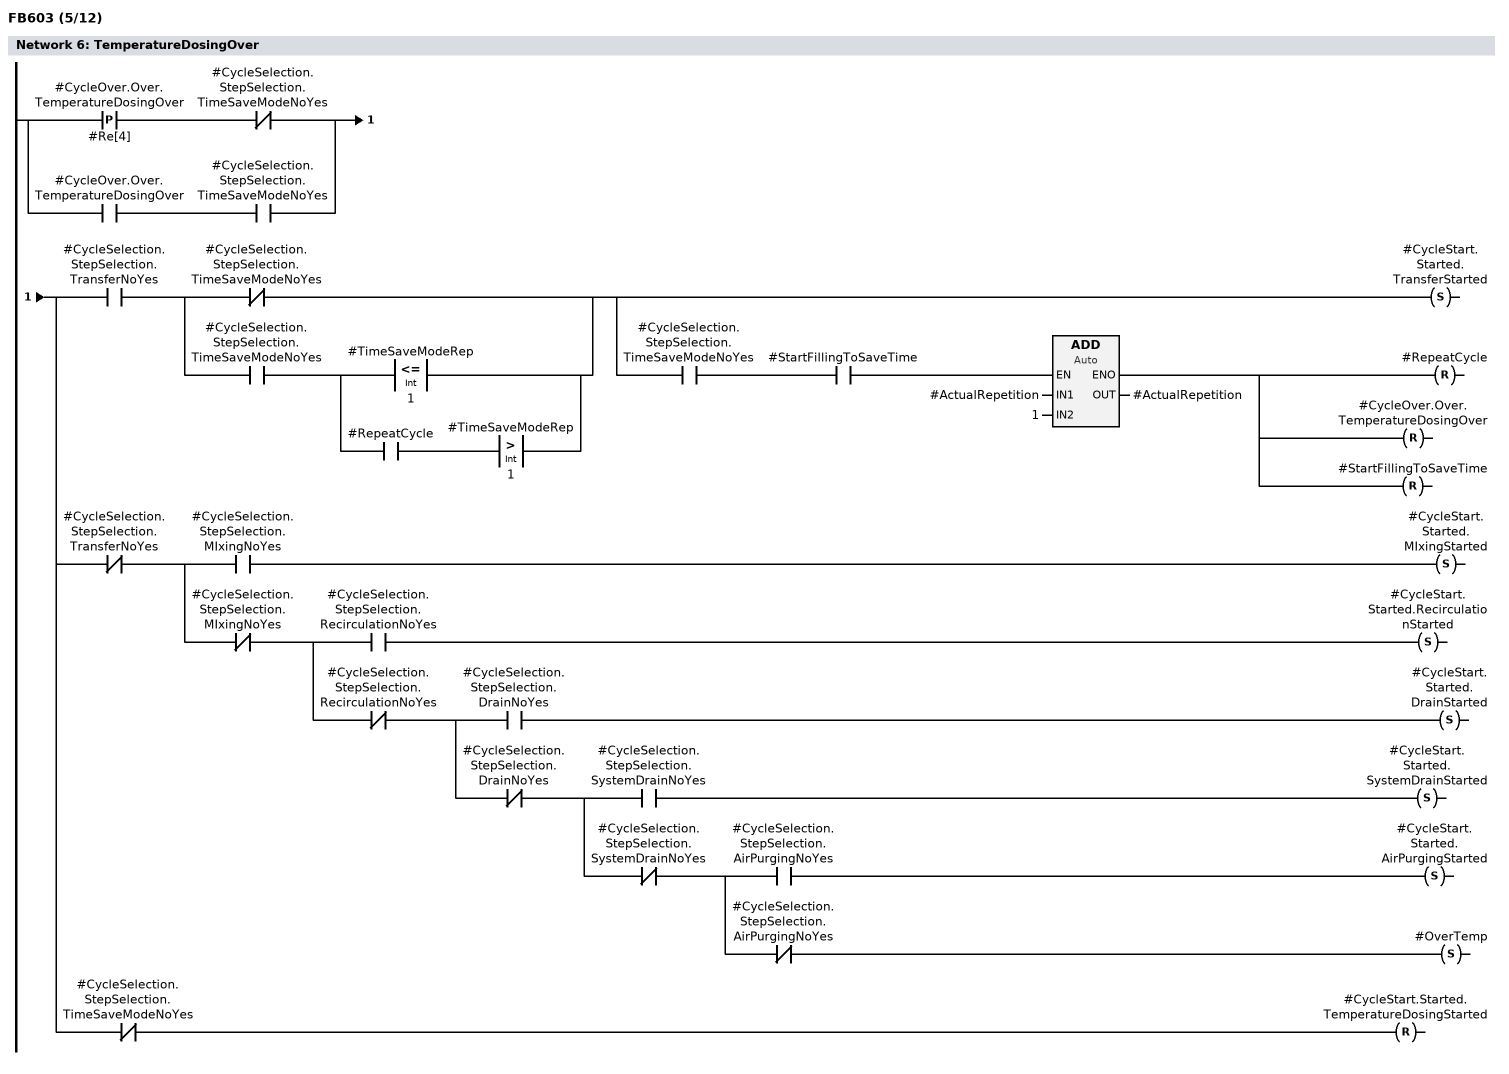
   RUNG wire#powerrail
      P_Contact(operand := #CycleOver.Over.TemperatureDosingOver, bit := #Re[4])
      I_Contact( #CycleSelection.StepSelection.TimeSaveModeNoYes )
      wire#w1
      Contact( #CycleSelection.StepSelection.TransferNoYes )
      wire#w2
      I_Contact( #CycleSelection.StepSelection.TimeSaveModeNoYes )
      wire#w3
      S_Coil( #CycleStart.Started.TransferStarted )
   END_RUNG
   RUNG wire#powerrail
      Contact( #CycleOver.Over.TemperatureDosingOver )
      Contact( #CycleSelection.StepSelection.TimeSaveModeNoYes )
   END_RUNG wire#w1
   RUNG wire#w2
      Contact( #CycleSelection.StepSelection.TimeSaveModeNoYes )
      wire#w4
      { S7_Templates := "SrcType := Int" } LE_Contact(in1 := #TimeSaveModeRep, in2 := 1)
   END_RUNG wire#w3
   RUNG wire#w4
      Contact( #RepeatCycle )
      { S7_Templates := "SrcType := Int" } GT_Contact(in1 := #TimeSaveModeRep, in2 := 1)
   END_RUNG wire#w3
   RUNG wire#w3
      Contact( #CycleSelection.StepSelection.TimeSaveModeNoYes )
      Contact( #StartFillingToSaveTime )
      Add(in1 := #ActualRepetition, in2 := 1, out => #ActualRepetition)
      wire#w5
      R_Coil( #RepeatCycle )
   END_RUNG
   RUNG wire#w5
      R_Coil( #CycleOver.Over.TemperatureDosingOver )
   END_RUNG
   RUNG wire#w5
      R_Coil( #StartFillingToSaveTime )
   END_RUNG
   RUNG wire#w1
      I_Contact( #CycleSelection.StepSelection.TransferNoYes )
      wire#w6
      Contact( #CycleSelection.StepSelection.MIxingNoYes )
      S_Coil( #CycleStart.Started.MIxingStarted )
   END_RUNG
   RUNG wire#w6
      I_Contact( #CycleSelection.StepSelection.MIxingNoYes )
      wire#w7
      Contact( #CycleSelection.StepSelection.RecirculationNoYes )
      S_Coil( #CycleStart.Started.RecirculationStarted )
   END_RUNG
   RUNG wire#w7
      I_Contact( #CycleSelection.StepSelection.RecirculationNoYes )
      wire#w8
      Contact( #CycleSelection.StepSelection.DrainNoYes )
      S_Coil( #CycleStart.Started.DrainStarted )
   END_RUNG
   RUNG wire#w8
      I_Contact( #CycleSelection.StepSelection.DrainNoYes )
      wire#w9
      Contact( #CycleSelection.StepSelection.SystemDrainNoYes )
      S_Coil( #CycleStart.Started.SystemDrainStarted )
   END_RUNG
   RUNG wire#w9
      I_Contact( #CycleSelection.StepSelection.SystemDrainNoYes )
      wire#w10
      Contact( #CycleSelection.StepSelection.AirPurgingNoYes )
      S_Coil( #CycleStart.Started.AirPurgingStarted )
   END_RUNG
   RUNG wire#w10
      I_Contact( #CycleSelection.StepSelection.AirPurgingNoYes )
      S_Coil( #OverTemp )
   END_RUNG
   RUNG wire#w1
      I_Contact( #CycleSelection.StepSelection.TimeSaveModeNoYes )
      R_Coil( #CycleStart.Started.TemperatureDosingStarted )
   END_RUNG
   // the same network as SCL:
   #_w1 := #CycleOver.Over.TemperatureDosingOver AND NOT #Re[4];   // rising edge of #CycleOver.Over.TemperatureDosingOver
   #Re[4] := #CycleOver.Over.TemperatureDosingOver;
   #_w2 := (#_w1 AND NOT #CycleSelection.StepSelection.TimeSaveModeNoYes) OR (#CycleOver.Over.TemperatureDosingOver AND #CycleSelection.StepSelection.TimeSaveModeNoYes);
   #_w3 := #_w2 AND #CycleSelection.StepSelection.TransferNoYes AND (NOT #CycleSelection.StepSelection.TimeSaveModeNoYes OR (#CycleSelection.StepSelection.TimeSaveModeNoYes AND ((#TimeSaveModeRep <= 1) OR (#RepeatCycle AND (#TimeSaveModeRep > 1)))));
   IF #_w3 THEN #CycleStart.Started.TransferStarted := TRUE; END_IF;
   IF #_w3 AND #CycleSelection.StepSelection.TimeSaveModeNoYes AND #StartFillingToSaveTime THEN
       #ActualRepetition := #ActualRepetition + 1;
       #RepeatCycle := FALSE;
       #CycleOver.Over.TemperatureDosingOver := FALSE;
       #StartFillingToSaveTime := FALSE;
   END_IF;
   #_w4 := #_w2 AND NOT #CycleSelection.StepSelection.TransferNoYes;
   IF #_w4 AND #CycleSelection.StepSelection.MIxingNoYes THEN
       #CycleStart.Started.MIxingStarted := TRUE;
   END_IF;
   #_w5 := #_w4 AND NOT #CycleSelection.StepSelection.MIxingNoYes;
   IF #_w5 AND #CycleSelection.StepSelection.RecirculationNoYes THEN
       #CycleStart.Started.RecirculationStarted := TRUE;
   END_IF;
   #_w6 := #_w5 AND NOT #CycleSelection.StepSelection.RecirculationNoYes;
   IF #_w6 AND #CycleSelection.StepSelection.DrainNoYes THEN
       #CycleStart.Started.DrainStarted := TRUE;
   END_IF;
   #_w7 := #_w6 AND NOT #CycleSelection.StepSelection.DrainNoYes;
   IF #_w7 AND #CycleSelection.StepSelection.SystemDrainNoYes THEN
       #CycleStart.Started.SystemDrainStarted := TRUE;
   END_IF;
   #_w8 := #_w7 AND NOT #CycleSelection.StepSelection.SystemDrainNoYes;
   IF #_w8 AND #CycleSelection.StepSelection.AirPurgingNoYes THEN
       #CycleStart.Started.AirPurgingStarted := TRUE;
   END_IF;
   IF #_w8 AND NOT #CycleSelection.StepSelection.AirPurgingNoYes THEN #OverTemp := TRUE; END_IF;
   IF #_w2 AND NOT #CycleSelection.StepSelection.TimeSaveModeNoYes THEN
       #CycleStart.Started.TemperatureDosingStarted := FALSE;
   END_IF;
END_REGION

REGION Network 7: TransferOver
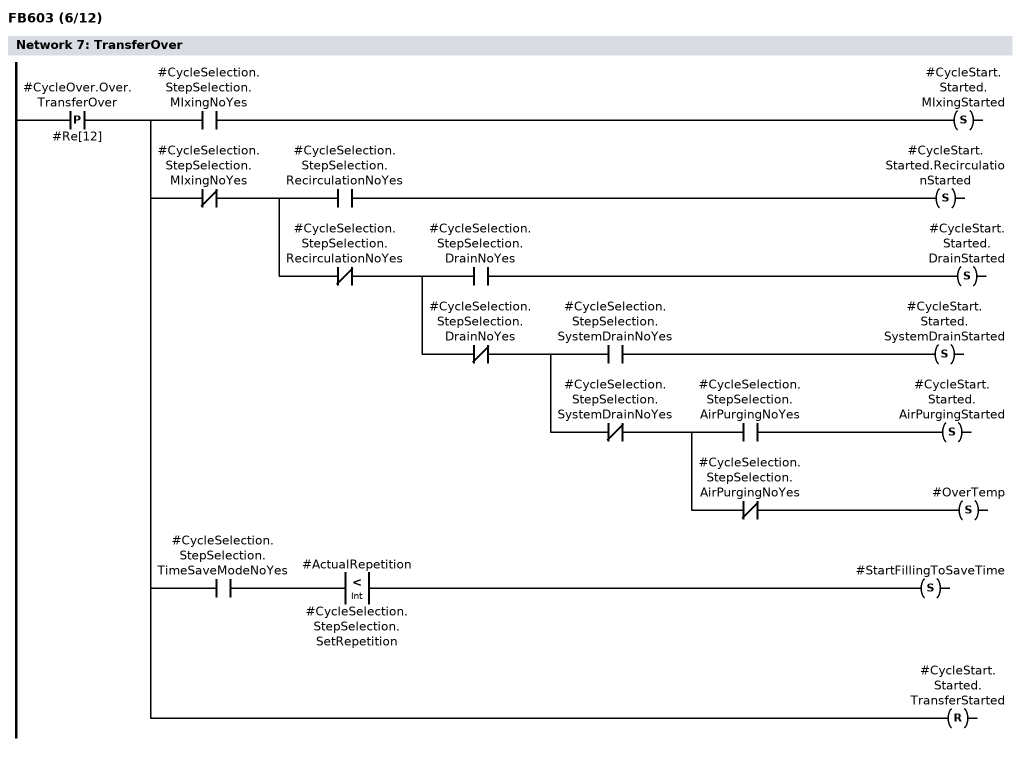
   RUNG wire#powerrail
      P_Contact(operand := #CycleOver.Over.TransferOver, bit := #Re[12])
      wire#w1
      Contact( #CycleSelection.StepSelection.MIxingNoYes )
      S_Coil( #CycleStart.Started.MIxingStarted )
   END_RUNG
   RUNG wire#w1
      I_Contact( #CycleSelection.StepSelection.MIxingNoYes )
      wire#w2
      Contact( #CycleSelection.StepSelection.RecirculationNoYes )
      S_Coil( #CycleStart.Started.RecirculationStarted )
   END_RUNG
   RUNG wire#w2
      I_Contact( #CycleSelection.StepSelection.RecirculationNoYes )
      wire#w3
      Contact( #CycleSelection.StepSelection.DrainNoYes )
      S_Coil( #CycleStart.Started.DrainStarted )
   END_RUNG
   RUNG wire#w3
      I_Contact( #CycleSelection.StepSelection.DrainNoYes )
      wire#w4
      Contact( #CycleSelection.StepSelection.SystemDrainNoYes )
      S_Coil( #CycleStart.Started.SystemDrainStarted )
   END_RUNG
   RUNG wire#w4
      I_Contact( #CycleSelection.StepSelection.SystemDrainNoYes )
      wire#w5
      Contact( #CycleSelection.StepSelection.AirPurgingNoYes )
      S_Coil( #CycleStart.Started.AirPurgingStarted )
   END_RUNG
   RUNG wire#w5
      I_Contact( #CycleSelection.StepSelection.AirPurgingNoYes )
      S_Coil( #OverTemp )
   END_RUNG
   RUNG wire#w1
      Contact( #CycleSelection.StepSelection.TimeSaveModeNoYes )
      { S7_Templates := "SrcType := Int" } LT_Contact(in1 := #ActualRepetition, in2 := #CycleSelection.StepSelection.SetRepetition)
      S_Coil( #StartFillingToSaveTime )
   END_RUNG
   RUNG wire#w1
      R_Coil( #CycleStart.Started.TransferStarted )
   END_RUNG
   // the same network as SCL:
   #_w1 := #CycleOver.Over.TransferOver AND NOT #Re[12];   // rising edge of #CycleOver.Over.TransferOver
   #Re[12] := #CycleOver.Over.TransferOver;
   IF #_w1 AND #CycleSelection.StepSelection.MIxingNoYes THEN
       #CycleStart.Started.MIxingStarted := TRUE;
   END_IF;
   #_w2 := #_w1 AND NOT #CycleSelection.StepSelection.MIxingNoYes;
   IF #_w2 AND #CycleSelection.StepSelection.RecirculationNoYes THEN
       #CycleStart.Started.RecirculationStarted := TRUE;
   END_IF;
   #_w3 := #_w2 AND NOT #CycleSelection.StepSelection.RecirculationNoYes;
   IF #_w3 AND #CycleSelection.StepSelection.DrainNoYes THEN
       #CycleStart.Started.DrainStarted := TRUE;
   END_IF;
   #_w4 := #_w3 AND NOT #CycleSelection.StepSelection.DrainNoYes;
   IF #_w4 AND #CycleSelection.StepSelection.SystemDrainNoYes THEN
       #CycleStart.Started.SystemDrainStarted := TRUE;
   END_IF;
   #_w5 := #_w4 AND NOT #CycleSelection.StepSelection.SystemDrainNoYes;
   IF #_w5 AND #CycleSelection.StepSelection.AirPurgingNoYes THEN
       #CycleStart.Started.AirPurgingStarted := TRUE;
   END_IF;
   IF #_w5 AND NOT #CycleSelection.StepSelection.AirPurgingNoYes THEN #OverTemp := TRUE; END_IF;
   IF #_w1 AND #CycleSelection.StepSelection.TimeSaveModeNoYes AND (#ActualRepetition < #CycleSelection.StepSelection.SetRepetition) THEN
       #StartFillingToSaveTime := TRUE;
   END_IF;
   IF #_w1 THEN #CycleStart.Started.TransferStarted := FALSE; END_IF;
END_REGION

REGION Network 8: TransferOver
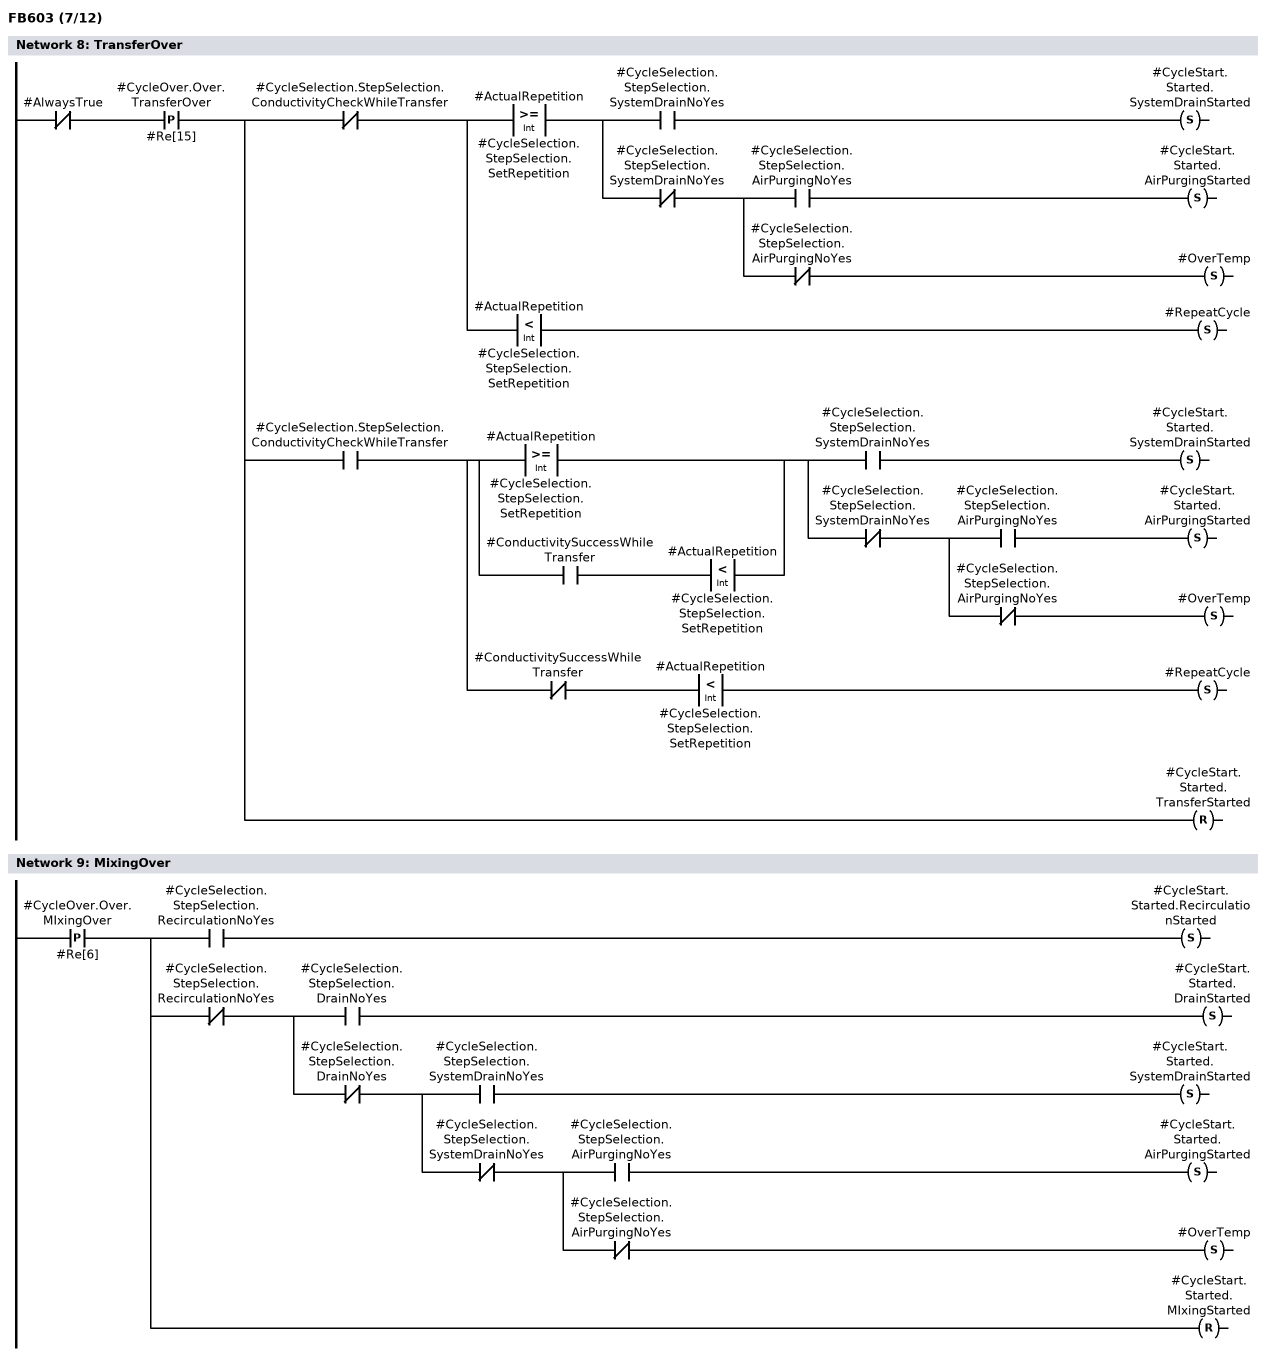
   RUNG wire#powerrail
      I_Contact( #AlwaysTrue )
      P_Contact(operand := #CycleOver.Over.TransferOver, bit := #Re[15])
      wire#w1
      I_Contact( #CycleSelection.StepSelection.ConductivityCheckWhileTransfer )
      wire#w2
      { S7_Templates := "SrcType := Int" } GE_Contact(in1 := #ActualRepetition, in2 := #CycleSelection.StepSelection.SetRepetition)
      wire#w3
      Contact( #CycleSelection.StepSelection.SystemDrainNoYes )
      S_Coil( #CycleStart.Started.SystemDrainStarted )
   END_RUNG
   RUNG wire#w3
      I_Contact( #CycleSelection.StepSelection.SystemDrainNoYes )
      wire#w4
      Contact( #CycleSelection.StepSelection.AirPurgingNoYes )
      S_Coil( #CycleStart.Started.AirPurgingStarted )
   END_RUNG
   RUNG wire#w4
      I_Contact( #CycleSelection.StepSelection.AirPurgingNoYes )
      S_Coil( #OverTemp )
   END_RUNG
   RUNG wire#w2
      { S7_Templates := "SrcType := Int" } LT_Contact(in1 := #ActualRepetition, in2 := #CycleSelection.StepSelection.SetRepetition)
      S_Coil( #RepeatCycle )
   END_RUNG
   RUNG wire#w1
      Contact( #CycleSelection.StepSelection.ConductivityCheckWhileTransfer )
      wire#w5
      { S7_Templates := "SrcType := Int" } GE_Contact(in1 := #ActualRepetition, in2 := #CycleSelection.StepSelection.SetRepetition)
      wire#w6
      Contact( #CycleSelection.StepSelection.SystemDrainNoYes )
      S_Coil( #CycleStart.Started.SystemDrainStarted )
   END_RUNG
   RUNG wire#w5
      Contact( #ConductivitySuccessWhileTransfer )
      { S7_Templates := "SrcType := Int" } LT_Contact(in1 := #ActualRepetition, in2 := #CycleSelection.StepSelection.SetRepetition)
   END_RUNG wire#w6
   RUNG wire#w6
      I_Contact( #CycleSelection.StepSelection.SystemDrainNoYes )
      wire#w7
      Contact( #CycleSelection.StepSelection.AirPurgingNoYes )
      S_Coil( #CycleStart.Started.AirPurgingStarted )
   END_RUNG
   RUNG wire#w7
      I_Contact( #CycleSelection.StepSelection.AirPurgingNoYes )
      S_Coil( #OverTemp )
   END_RUNG
   RUNG wire#w5
      I_Contact( #ConductivitySuccessWhileTransfer )
      { S7_Templates := "SrcType := Int" } LT_Contact(in1 := #ActualRepetition, in2 := #CycleSelection.StepSelection.SetRepetition)
      S_Coil( #RepeatCycle )
   END_RUNG
   RUNG wire#w1
      R_Coil( #CycleStart.Started.TransferStarted )
   END_RUNG
   // the same network as SCL:
   #_w1 := NOT #AlwaysTrue AND #CycleOver.Over.TransferOver AND NOT #Re[15];   // rising edge of #CycleOver.Over.TransferOver
   #Re[15] := #CycleOver.Over.TransferOver;
   #_w2 := #_w1 AND NOT #CycleSelection.StepSelection.ConductivityCheckWhileTransfer;
   #_w3 := #_w2 AND (#ActualRepetition >= #CycleSelection.StepSelection.SetRepetition);
   IF #_w3 AND #CycleSelection.StepSelection.SystemDrainNoYes THEN
       #CycleStart.Started.SystemDrainStarted := TRUE;
   END_IF;
   #_w4 := #_w3 AND NOT #CycleSelection.StepSelection.SystemDrainNoYes;
   IF #_w4 AND #CycleSelection.StepSelection.AirPurgingNoYes THEN
       #CycleStart.Started.AirPurgingStarted := TRUE;
   END_IF;
   IF #_w4 AND NOT #CycleSelection.StepSelection.AirPurgingNoYes THEN #OverTemp := TRUE; END_IF;
   IF #_w2 AND (#ActualRepetition < #CycleSelection.StepSelection.SetRepetition) THEN
       #RepeatCycle := TRUE;
   END_IF;
   #_w5 := #_w1 AND #CycleSelection.StepSelection.ConductivityCheckWhileTransfer;
   #_w6 := #_w5 AND ((#ActualRepetition >= #CycleSelection.StepSelection.SetRepetition) OR (#ConductivitySuccessWhileTransfer AND (#ActualRepetition < #CycleSelection.StepSelection.SetRepetition)));
   IF #_w6 AND #CycleSelection.StepSelection.SystemDrainNoYes THEN
       #CycleStart.Started.SystemDrainStarted := TRUE;
   END_IF;
   #_w7 := #_w6 AND NOT #CycleSelection.StepSelection.SystemDrainNoYes;
   IF #_w7 AND #CycleSelection.StepSelection.AirPurgingNoYes THEN
       #CycleStart.Started.AirPurgingStarted := TRUE;
   END_IF;
   IF #_w7 AND NOT #CycleSelection.StepSelection.AirPurgingNoYes THEN #OverTemp := TRUE; END_IF;
   IF #_w5 AND NOT #ConductivitySuccessWhileTransfer AND (#ActualRepetition < #CycleSelection.StepSelection.SetRepetition) THEN
       #RepeatCycle := TRUE;
   END_IF;
   IF #_w1 THEN #CycleStart.Started.TransferStarted := FALSE; END_IF;
END_REGION

REGION Network 9: MixingOver
   RUNG wire#powerrail
      P_Contact(operand := #CycleOver.Over.MIxingOver, bit := #Re[6])
      wire#w1
      Contact( #CycleSelection.StepSelection.RecirculationNoYes )
      S_Coil( #CycleStart.Started.RecirculationStarted )
   END_RUNG
   RUNG wire#w1
      I_Contact( #CycleSelection.StepSelection.RecirculationNoYes )
      wire#w2
      Contact( #CycleSelection.StepSelection.DrainNoYes )
      S_Coil( #CycleStart.Started.DrainStarted )
   END_RUNG
   RUNG wire#w2
      I_Contact( #CycleSelection.StepSelection.DrainNoYes )
      wire#w3
      Contact( #CycleSelection.StepSelection.SystemDrainNoYes )
      S_Coil( #CycleStart.Started.SystemDrainStarted )
   END_RUNG
   RUNG wire#w3
      I_Contact( #CycleSelection.StepSelection.SystemDrainNoYes )
      wire#w4
      Contact( #CycleSelection.StepSelection.AirPurgingNoYes )
      S_Coil( #CycleStart.Started.AirPurgingStarted )
   END_RUNG
   RUNG wire#w4
      I_Contact( #CycleSelection.StepSelection.AirPurgingNoYes )
      S_Coil( #OverTemp )
   END_RUNG
   RUNG wire#w1
      R_Coil( #CycleStart.Started.MIxingStarted )
   END_RUNG
   // the same network as SCL:
   #_w1 := #CycleOver.Over.MIxingOver AND NOT #Re[6];   // rising edge of #CycleOver.Over.MIxingOver
   #Re[6] := #CycleOver.Over.MIxingOver;
   IF #_w1 AND #CycleSelection.StepSelection.RecirculationNoYes THEN
       #CycleStart.Started.RecirculationStarted := TRUE;
   END_IF;
   #_w2 := #_w1 AND NOT #CycleSelection.StepSelection.RecirculationNoYes;
   IF #_w2 AND #CycleSelection.StepSelection.DrainNoYes THEN
       #CycleStart.Started.DrainStarted := TRUE;
   END_IF;
   #_w3 := #_w2 AND NOT #CycleSelection.StepSelection.DrainNoYes;
   IF #_w3 AND #CycleSelection.StepSelection.SystemDrainNoYes THEN
       #CycleStart.Started.SystemDrainStarted := TRUE;
   END_IF;
   #_w4 := #_w3 AND NOT #CycleSelection.StepSelection.SystemDrainNoYes;
   IF #_w4 AND #CycleSelection.StepSelection.AirPurgingNoYes THEN
       #CycleStart.Started.AirPurgingStarted := TRUE;
   END_IF;
   IF #_w4 AND NOT #CycleSelection.StepSelection.AirPurgingNoYes THEN #OverTemp := TRUE; END_IF;
   IF #_w1 THEN #CycleStart.Started.MIxingStarted := FALSE; END_IF;
END_REGION

REGION Network 10: RecirculationOver
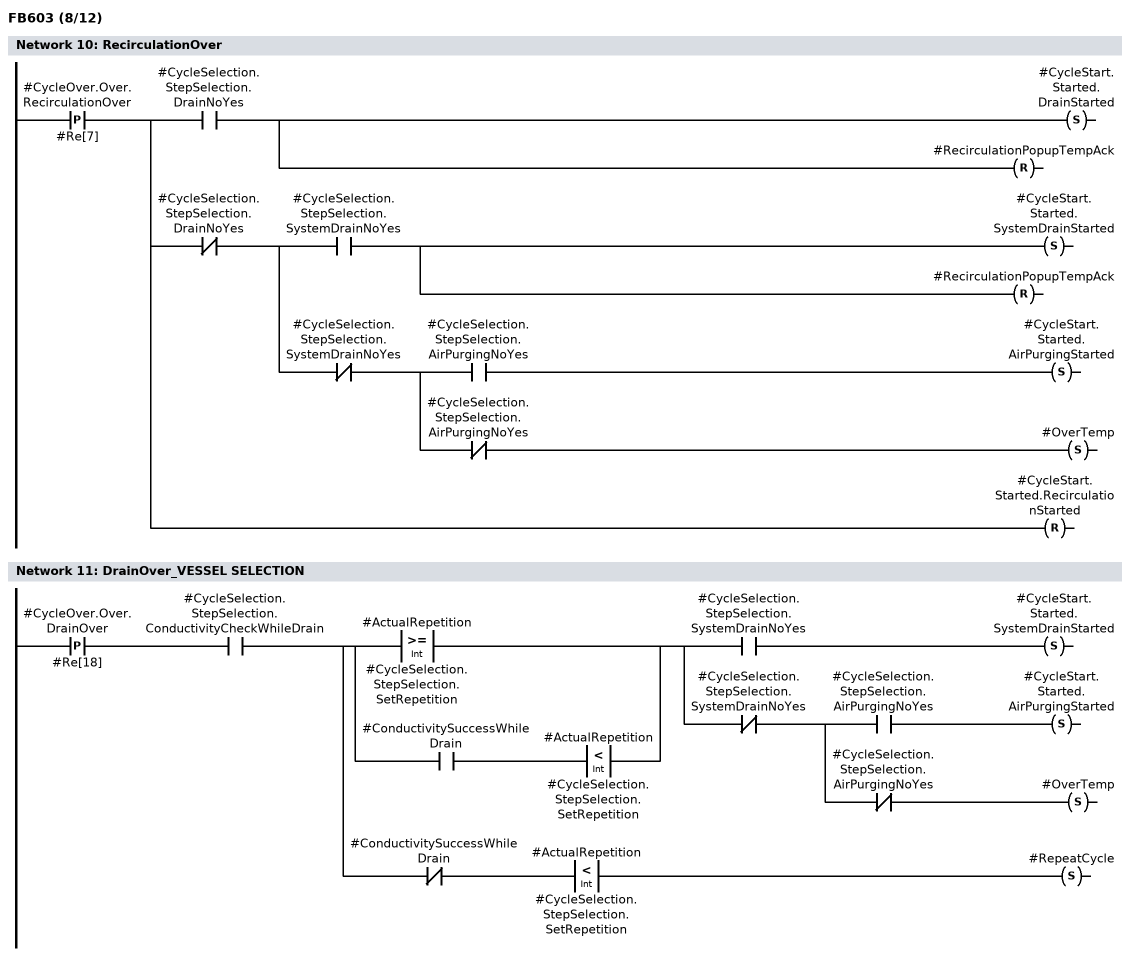
   RUNG wire#powerrail
      P_Contact(operand := #CycleOver.Over.RecirculationOver, bit := #Re[7])
      wire#w1
      Contact( #CycleSelection.StepSelection.DrainNoYes )
      wire#w2
      S_Coil( #CycleStart.Started.DrainStarted )
   END_RUNG
   RUNG wire#w2
      R_Coil( #RecirculationPopupTempAck )
   END_RUNG
   RUNG wire#w1
      I_Contact( #CycleSelection.StepSelection.DrainNoYes )
      wire#w3
      Contact( #CycleSelection.StepSelection.SystemDrainNoYes )
      wire#w4
      S_Coil( #CycleStart.Started.SystemDrainStarted )
   END_RUNG
   RUNG wire#w4
      R_Coil( #RecirculationPopupTempAck )
   END_RUNG
   RUNG wire#w3
      I_Contact( #CycleSelection.StepSelection.SystemDrainNoYes )
      wire#w5
      Contact( #CycleSelection.StepSelection.AirPurgingNoYes )
      S_Coil( #CycleStart.Started.AirPurgingStarted )
   END_RUNG
   RUNG wire#w5
      I_Contact( #CycleSelection.StepSelection.AirPurgingNoYes )
      S_Coil( #OverTemp )
   END_RUNG
   RUNG wire#w1
      R_Coil( #CycleStart.Started.RecirculationStarted )
   END_RUNG
   // the same network as SCL:
   #_w1 := #CycleOver.Over.RecirculationOver AND NOT #Re[7];   // rising edge of #CycleOver.Over.RecirculationOver
   #Re[7] := #CycleOver.Over.RecirculationOver;
   IF #_w1 AND #CycleSelection.StepSelection.DrainNoYes THEN
       #CycleStart.Started.DrainStarted := TRUE;
       #RecirculationPopupTempAck := FALSE;
   END_IF;
   #_w2 := #_w1 AND NOT #CycleSelection.StepSelection.DrainNoYes;
   IF #_w2 AND #CycleSelection.StepSelection.SystemDrainNoYes THEN
       #CycleStart.Started.SystemDrainStarted := TRUE;
       #RecirculationPopupTempAck := FALSE;
   END_IF;
   #_w3 := #_w2 AND NOT #CycleSelection.StepSelection.SystemDrainNoYes;
   IF #_w3 AND #CycleSelection.StepSelection.AirPurgingNoYes THEN
       #CycleStart.Started.AirPurgingStarted := TRUE;
   END_IF;
   IF #_w3 AND NOT #CycleSelection.StepSelection.AirPurgingNoYes THEN #OverTemp := TRUE; END_IF;
   IF #_w1 THEN #CycleStart.Started.RecirculationStarted := FALSE; END_IF;
END_REGION

REGION Network 11: DrainOver_VESSEL SELECTION
   RUNG wire#powerrail
      P_Contact(operand := #CycleOver.Over.DrainOver, bit := #Re[18])
      Contact( #CycleSelection.StepSelection.ConductivityCheckWhileDrain )
      wire#w1
      { S7_Templates := "SrcType := Int" } GE_Contact(in1 := #ActualRepetition, in2 := #CycleSelection.StepSelection.SetRepetition)
      wire#w2
      Contact( #CycleSelection.StepSelection.SystemDrainNoYes )
      S_Coil( #CycleStart.Started.SystemDrainStarted )
   END_RUNG
   RUNG wire#w1
      Contact( #ConductivitySuccessWhileDrain )
      { S7_Templates := "SrcType := Int" } LT_Contact(in1 := #ActualRepetition, in2 := #CycleSelection.StepSelection.SetRepetition)
   END_RUNG wire#w2
   RUNG wire#w2
      I_Contact( #CycleSelection.StepSelection.SystemDrainNoYes )
      wire#w3
      Contact( #CycleSelection.StepSelection.AirPurgingNoYes )
      S_Coil( #CycleStart.Started.AirPurgingStarted )
   END_RUNG
   RUNG wire#w3
      I_Contact( #CycleSelection.StepSelection.AirPurgingNoYes )
      S_Coil( #OverTemp )
   END_RUNG
   RUNG wire#w1
      I_Contact( #ConductivitySuccessWhileDrain )
      { S7_Templates := "SrcType := Int" } LT_Contact(in1 := #ActualRepetition, in2 := #CycleSelection.StepSelection.SetRepetition)
      S_Coil( #RepeatCycle )
   END_RUNG
   // the same network as SCL:
   #_w1 := #CycleOver.Over.DrainOver AND NOT #Re[18];   // rising edge of #CycleOver.Over.DrainOver
   #Re[18] := #CycleOver.Over.DrainOver;
   #_w2 := #_w1 AND #CycleSelection.StepSelection.ConductivityCheckWhileDrain;
   #_w3 := #_w2 AND ((#ActualRepetition >= #CycleSelection.StepSelection.SetRepetition) OR (#ConductivitySuccessWhileDrain AND (#ActualRepetition < #CycleSelection.StepSelection.SetRepetition)));
   IF #_w3 AND #CycleSelection.StepSelection.SystemDrainNoYes THEN
       #CycleStart.Started.SystemDrainStarted := TRUE;
   END_IF;
   #_w4 := #_w3 AND NOT #CycleSelection.StepSelection.SystemDrainNoYes;
   IF #_w4 AND #CycleSelection.StepSelection.AirPurgingNoYes THEN
       #CycleStart.Started.AirPurgingStarted := TRUE;
   END_IF;
   IF #_w4 AND NOT #CycleSelection.StepSelection.AirPurgingNoYes THEN #OverTemp := TRUE; END_IF;
   IF #_w2 AND NOT #ConductivitySuccessWhileDrain AND (#ActualRepetition < #CycleSelection.StepSelection.SetRepetition) THEN
       #RepeatCycle := TRUE;
   END_IF;
END_REGION

REGION Network 12: DRAIN OVER (WITHOUT CONDUCTIVITY SEL.)
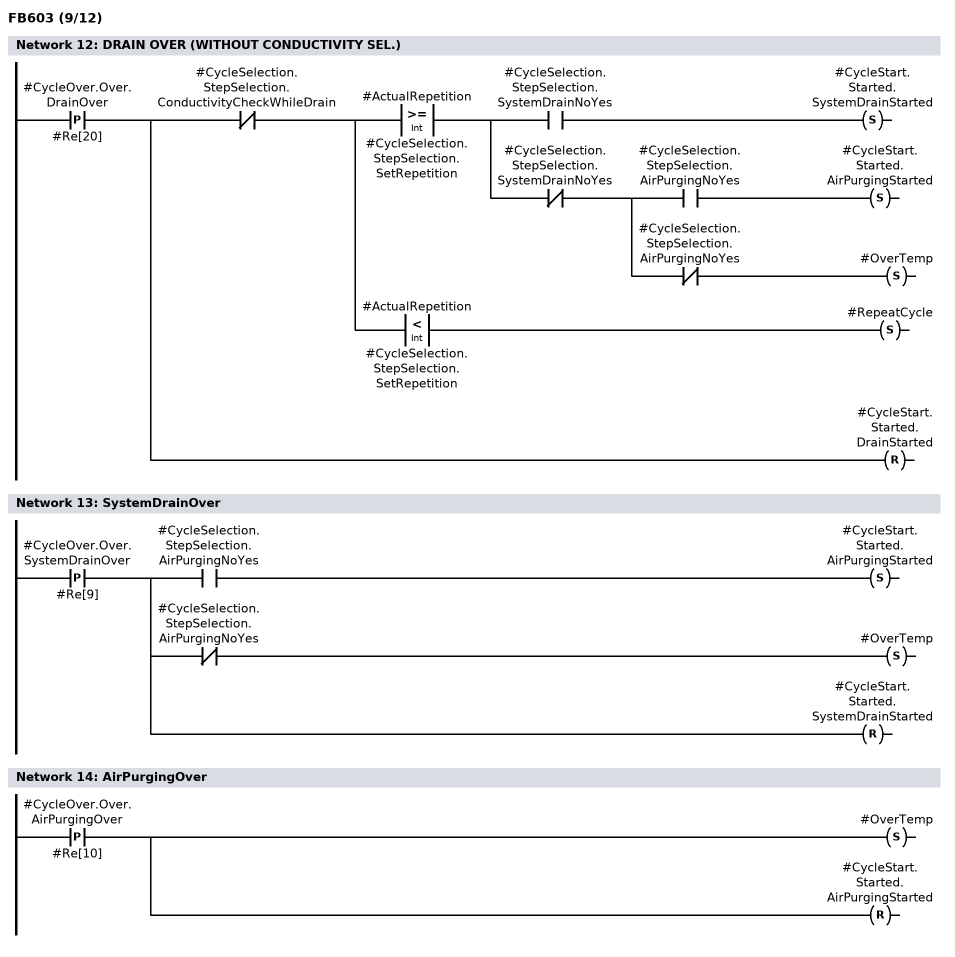
   RUNG wire#powerrail
      P_Contact(operand := #CycleOver.Over.DrainOver, bit := #Re[20])
      wire#w1
      I_Contact( #CycleSelection.StepSelection.ConductivityCheckWhileDrain )
      wire#w2
      { S7_Templates := "SrcType := Int" } GE_Contact(in1 := #ActualRepetition, in2 := #CycleSelection.StepSelection.SetRepetition)
      wire#w3
      Contact( #CycleSelection.StepSelection.SystemDrainNoYes )
      S_Coil( #CycleStart.Started.SystemDrainStarted )
   END_RUNG
   RUNG wire#w3
      I_Contact( #CycleSelection.StepSelection.SystemDrainNoYes )
      wire#w4
      Contact( #CycleSelection.StepSelection.AirPurgingNoYes )
      S_Coil( #CycleStart.Started.AirPurgingStarted )
   END_RUNG
   RUNG wire#w4
      I_Contact( #CycleSelection.StepSelection.AirPurgingNoYes )
      S_Coil( #OverTemp )
   END_RUNG
   RUNG wire#w2
      { S7_Templates := "SrcType := Int" } LT_Contact(in1 := #ActualRepetition, in2 := #CycleSelection.StepSelection.SetRepetition)
      S_Coil( #RepeatCycle )
   END_RUNG
   RUNG wire#w1
      R_Coil( #CycleStart.Started.DrainStarted )
   END_RUNG
   // the same network as SCL:
   #_w1 := #CycleOver.Over.DrainOver AND NOT #Re[20];   // rising edge of #CycleOver.Over.DrainOver
   #Re[20] := #CycleOver.Over.DrainOver;
   #_w2 := #_w1 AND NOT #CycleSelection.StepSelection.ConductivityCheckWhileDrain;
   #_w3 := #_w2 AND (#ActualRepetition >= #CycleSelection.StepSelection.SetRepetition);
   IF #_w3 AND #CycleSelection.StepSelection.SystemDrainNoYes THEN
       #CycleStart.Started.SystemDrainStarted := TRUE;
   END_IF;
   #_w4 := #_w3 AND NOT #CycleSelection.StepSelection.SystemDrainNoYes;
   IF #_w4 AND #CycleSelection.StepSelection.AirPurgingNoYes THEN
       #CycleStart.Started.AirPurgingStarted := TRUE;
   END_IF;
   IF #_w4 AND NOT #CycleSelection.StepSelection.AirPurgingNoYes THEN #OverTemp := TRUE; END_IF;
   IF #_w2 AND (#ActualRepetition < #CycleSelection.StepSelection.SetRepetition) THEN
       #RepeatCycle := TRUE;
   END_IF;
   IF #_w1 THEN #CycleStart.Started.DrainStarted := FALSE; END_IF;
END_REGION

REGION Network 13: SystemDrainOver
   RUNG wire#powerrail
      P_Contact(operand := #CycleOver.Over.SystemDrainOver, bit := #Re[9])
      wire#w1
      Contact( #CycleSelection.StepSelection.AirPurgingNoYes )
      S_Coil( #CycleStart.Started.AirPurgingStarted )
   END_RUNG
   RUNG wire#w1
      I_Contact( #CycleSelection.StepSelection.AirPurgingNoYes )
      S_Coil( #OverTemp )
   END_RUNG
   RUNG wire#w1
      R_Coil( #CycleStart.Started.SystemDrainStarted )
   END_RUNG
   // the same network as SCL:
   #_w1 := #CycleOver.Over.SystemDrainOver AND NOT #Re[9];   // rising edge of #CycleOver.Over.SystemDrainOver
   #Re[9] := #CycleOver.Over.SystemDrainOver;
   IF #_w1 AND #CycleSelection.StepSelection.AirPurgingNoYes THEN
       #CycleStart.Started.AirPurgingStarted := TRUE;
   END_IF;
   IF #_w1 AND NOT #CycleSelection.StepSelection.AirPurgingNoYes THEN #OverTemp := TRUE; END_IF;
   IF #_w1 THEN #CycleStart.Started.SystemDrainStarted := FALSE; END_IF;
END_REGION

REGION Network 14: AirPurgingOver
   RUNG wire#powerrail
      P_Contact(operand := #CycleOver.Over.AirPurgingOver, bit := #Re[10])
      wire#w1
      S_Coil( #OverTemp )
   END_RUNG
   RUNG wire#w1
      R_Coil( #CycleStart.Started.AirPurgingStarted )
   END_RUNG
   // the same network as SCL:
   #_w1 := #CycleOver.Over.AirPurgingOver AND NOT #Re[10];   // rising edge of #CycleOver.Over.AirPurgingOver
   #Re[10] := #CycleOver.Over.AirPurgingOver;
   IF #_w1 THEN
       #OverTemp := TRUE;
       #CycleStart.Started.AirPurgingStarted := FALSE;
   END_IF;
END_REGION

REGION Network 15: Reset
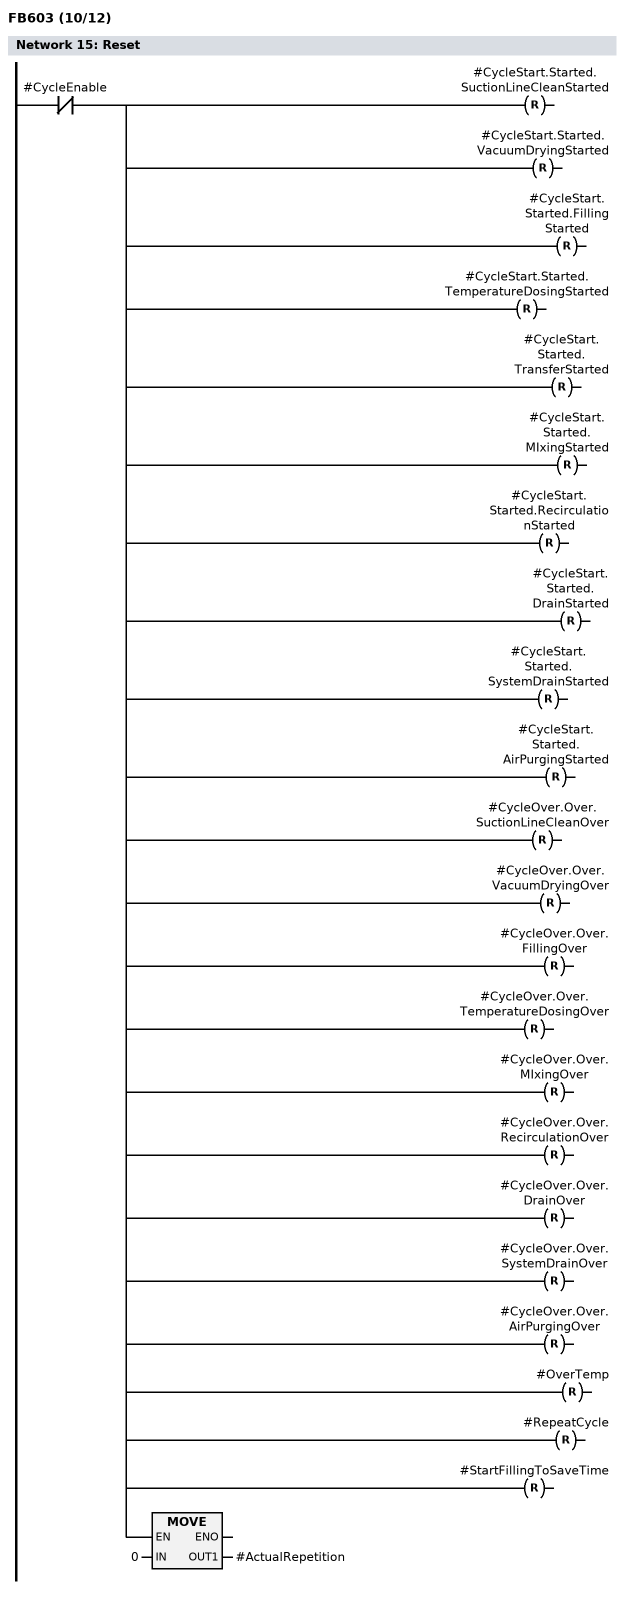
   RUNG wire#powerrail
      I_Contact( #CycleEnable )
      wire#w1
      R_Coil( #CycleStart.Started.SuctionLineCleanStarted )
   END_RUNG
   RUNG wire#w1
      R_Coil( #CycleStart.Started.VacuumDryingStarted )
   END_RUNG
   RUNG wire#w1
      R_Coil( #CycleStart.Started.FillingStarted )
   END_RUNG
   RUNG wire#w1
      R_Coil( #CycleStart.Started.TemperatureDosingStarted )
   END_RUNG
   RUNG wire#w1
      R_Coil( #CycleStart.Started.TransferStarted )
   END_RUNG
   RUNG wire#w1
      R_Coil( #CycleStart.Started.MIxingStarted )
   END_RUNG
   RUNG wire#w1
      R_Coil( #CycleStart.Started.RecirculationStarted )
   END_RUNG
   RUNG wire#w1
      R_Coil( #CycleStart.Started.DrainStarted )
   END_RUNG
   RUNG wire#w1
      R_Coil( #CycleStart.Started.SystemDrainStarted )
   END_RUNG
   RUNG wire#w1
      R_Coil( #CycleStart.Started.AirPurgingStarted )
   END_RUNG
   RUNG wire#w1
      R_Coil( #CycleOver.Over.SuctionLineCleanOver )
   END_RUNG
   RUNG wire#w1
      R_Coil( #CycleOver.Over.VacuumDryingOver )
   END_RUNG
   RUNG wire#w1
      R_Coil( #CycleOver.Over.FillingOver )
   END_RUNG
   RUNG wire#w1
      R_Coil( #CycleOver.Over.TemperatureDosingOver )
   END_RUNG
   RUNG wire#w1
      R_Coil( #CycleOver.Over.MIxingOver )
   END_RUNG
   RUNG wire#w1
      R_Coil( #CycleOver.Over.RecirculationOver )
   END_RUNG
   RUNG wire#w1
      R_Coil( #CycleOver.Over.DrainOver )
   END_RUNG
   RUNG wire#w1
      R_Coil( #CycleOver.Over.SystemDrainOver )
   END_RUNG
   RUNG wire#w1
      R_Coil( #CycleOver.Over.AirPurgingOver )
   END_RUNG
   RUNG wire#w1
      R_Coil( #OverTemp )
   END_RUNG
   RUNG wire#w1
      R_Coil( #RepeatCycle )
   END_RUNG
   RUNG wire#w1
      R_Coil( #StartFillingToSaveTime )
   END_RUNG
   RUNG wire#w1
      Move(in := 0, out1 => #ActualRepetition)
   END_RUNG
   // the same network as SCL:
   IF NOT #CycleEnable THEN
       #CycleStart.Started.SuctionLineCleanStarted := FALSE;
       #CycleStart.Started.VacuumDryingStarted := FALSE;
       #CycleStart.Started.FillingStarted := FALSE;
       #CycleStart.Started.TemperatureDosingStarted := FALSE;
       #CycleStart.Started.TransferStarted := FALSE;
       #CycleStart.Started.MIxingStarted := FALSE;
       #CycleStart.Started.RecirculationStarted := FALSE;
       #CycleStart.Started.DrainStarted := FALSE;
       #CycleStart.Started.SystemDrainStarted := FALSE;
       #CycleStart.Started.AirPurgingStarted := FALSE;
       #CycleOver.Over.SuctionLineCleanOver := FALSE;
       #CycleOver.Over.VacuumDryingOver := FALSE;
       #CycleOver.Over.FillingOver := FALSE;
       #CycleOver.Over.TemperatureDosingOver := FALSE;
       #CycleOver.Over.MIxingOver := FALSE;
       #CycleOver.Over.RecirculationOver := FALSE;
       #CycleOver.Over.DrainOver := FALSE;
       #CycleOver.Over.SystemDrainOver := FALSE;
       #CycleOver.Over.AirPurgingOver := FALSE;
       #OverTemp := FALSE;
       #RepeatCycle := FALSE;
       #StartFillingToSaveTime := FALSE;
       #ActualRepetition := 0;
   END_IF;
END_REGION

REGION Network 16: Reset
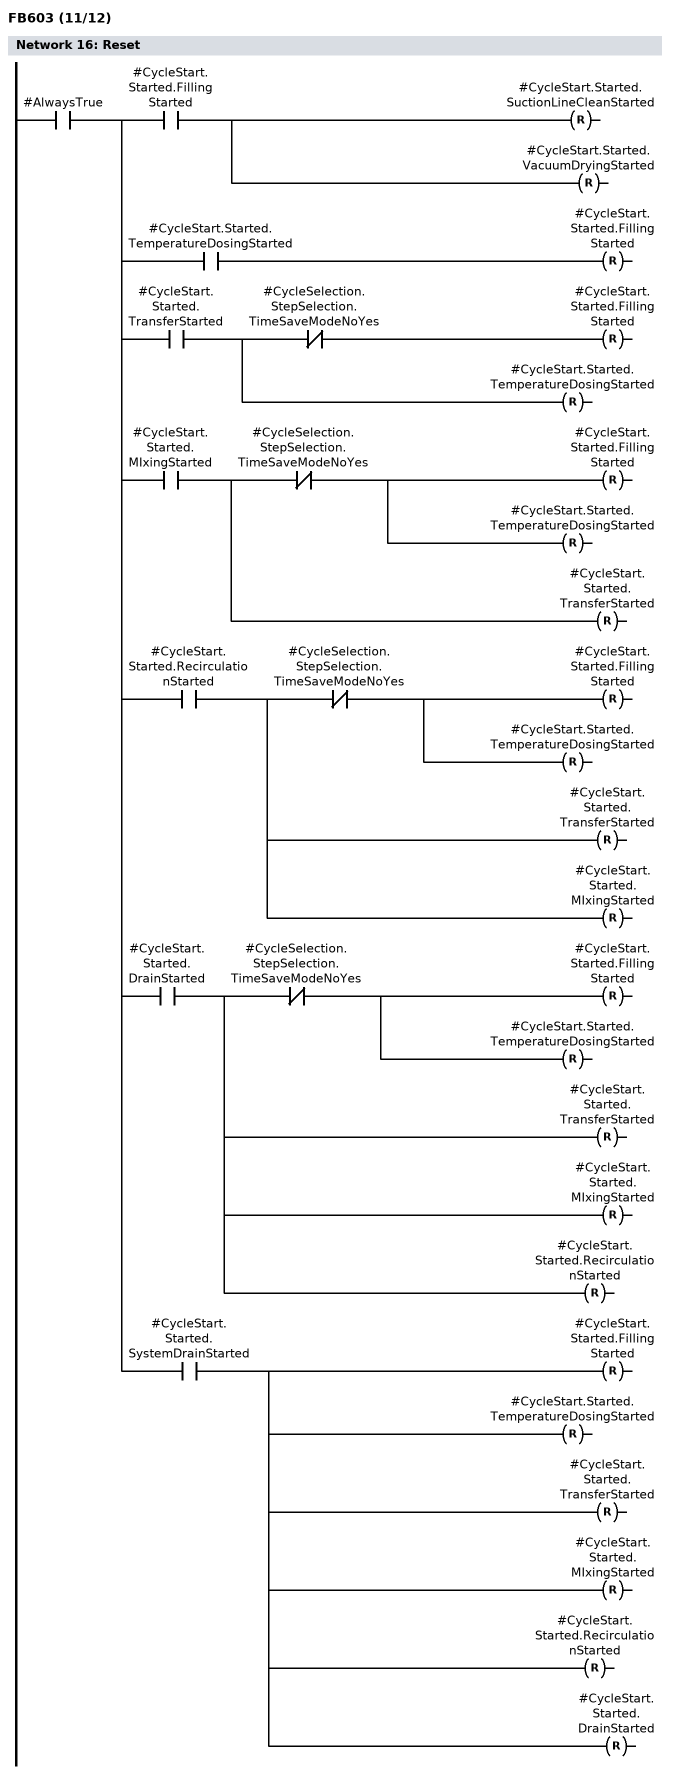
   RUNG wire#powerrail
      Contact( #AlwaysTrue )
      wire#w1
      Contact( #CycleStart.Started.FillingStarted )
      wire#w2
      R_Coil( #CycleStart.Started.SuctionLineCleanStarted )
   END_RUNG
   RUNG wire#w2
      R_Coil( #CycleStart.Started.VacuumDryingStarted )
   END_RUNG
   RUNG wire#w1
      Contact( #CycleStart.Started.TemperatureDosingStarted )
      R_Coil( #CycleStart.Started.FillingStarted )
   END_RUNG
   RUNG wire#w1
      Contact( #CycleStart.Started.TransferStarted )
      wire#w3
      I_Contact( #CycleSelection.StepSelection.TimeSaveModeNoYes )
      R_Coil( #CycleStart.Started.FillingStarted )
   END_RUNG
   RUNG wire#w3
      R_Coil( #CycleStart.Started.TemperatureDosingStarted )
   END_RUNG
   RUNG wire#w1
      Contact( #CycleStart.Started.MIxingStarted )
      wire#w4
      I_Contact( #CycleSelection.StepSelection.TimeSaveModeNoYes )
      wire#w5
      R_Coil( #CycleStart.Started.FillingStarted )
   END_RUNG
   RUNG wire#w5
      R_Coil( #CycleStart.Started.TemperatureDosingStarted )
   END_RUNG
   RUNG wire#w4
      R_Coil( #CycleStart.Started.TransferStarted )
   END_RUNG
   RUNG wire#w1
      Contact( #CycleStart.Started.RecirculationStarted )
      wire#w6
      I_Contact( #CycleSelection.StepSelection.TimeSaveModeNoYes )
      wire#w7
      R_Coil( #CycleStart.Started.FillingStarted )
   END_RUNG
   RUNG wire#w7
      R_Coil( #CycleStart.Started.TemperatureDosingStarted )
   END_RUNG
   RUNG wire#w6
      R_Coil( #CycleStart.Started.TransferStarted )
   END_RUNG
   RUNG wire#w6
      R_Coil( #CycleStart.Started.MIxingStarted )
   END_RUNG
   RUNG wire#w1
      Contact( #CycleStart.Started.DrainStarted )
      wire#w8
      I_Contact( #CycleSelection.StepSelection.TimeSaveModeNoYes )
      wire#w9
      R_Coil( #CycleStart.Started.FillingStarted )
   END_RUNG
   RUNG wire#w9
      R_Coil( #CycleStart.Started.TemperatureDosingStarted )
   END_RUNG
   RUNG wire#w8
      R_Coil( #CycleStart.Started.TransferStarted )
   END_RUNG
   RUNG wire#w8
      R_Coil( #CycleStart.Started.MIxingStarted )
   END_RUNG
   RUNG wire#w8
      R_Coil( #CycleStart.Started.RecirculationStarted )
   END_RUNG
   RUNG wire#w1
      Contact( #CycleStart.Started.SystemDrainStarted )
      wire#w10
      R_Coil( #CycleStart.Started.FillingStarted )
   END_RUNG
   RUNG wire#w10
      R_Coil( #CycleStart.Started.TemperatureDosingStarted )
   END_RUNG
   RUNG wire#w10
      R_Coil( #CycleStart.Started.TransferStarted )
   END_RUNG
   RUNG wire#w10
      R_Coil( #CycleStart.Started.MIxingStarted )
   END_RUNG
   RUNG wire#w10
      R_Coil( #CycleStart.Started.RecirculationStarted )
   END_RUNG
   RUNG wire#w10
      R_Coil( #CycleStart.Started.DrainStarted )
   END_RUNG
   // the same network as SCL:
   IF #AlwaysTrue AND #CycleStart.Started.FillingStarted THEN
       #CycleStart.Started.SuctionLineCleanStarted := FALSE;
       #CycleStart.Started.VacuumDryingStarted := FALSE;
   END_IF;
   IF #AlwaysTrue AND #CycleStart.Started.TemperatureDosingStarted THEN
       #CycleStart.Started.FillingStarted := FALSE;
   END_IF;
   #_w1 := #AlwaysTrue AND #CycleStart.Started.TransferStarted;
   IF #_w1 AND NOT #CycleSelection.StepSelection.TimeSaveModeNoYes THEN
       #CycleStart.Started.FillingStarted := FALSE;
   END_IF;
   IF #_w1 THEN #CycleStart.Started.TemperatureDosingStarted := FALSE; END_IF;
   #_w2 := #AlwaysTrue AND #CycleStart.Started.MIxingStarted;
   IF #_w2 AND NOT #CycleSelection.StepSelection.TimeSaveModeNoYes THEN
       #CycleStart.Started.FillingStarted := FALSE;
       #CycleStart.Started.TemperatureDosingStarted := FALSE;
   END_IF;
   IF #_w2 THEN #CycleStart.Started.TransferStarted := FALSE; END_IF;
   #_w3 := #AlwaysTrue AND #CycleStart.Started.RecirculationStarted;
   IF #_w3 AND NOT #CycleSelection.StepSelection.TimeSaveModeNoYes THEN
       #CycleStart.Started.FillingStarted := FALSE;
       #CycleStart.Started.TemperatureDosingStarted := FALSE;
   END_IF;
   IF #_w3 THEN
       #CycleStart.Started.TransferStarted := FALSE;
       #CycleStart.Started.MIxingStarted := FALSE;
   END_IF;
   #_w4 := #AlwaysTrue AND #CycleStart.Started.DrainStarted;
   IF #_w4 AND NOT #CycleSelection.StepSelection.TimeSaveModeNoYes THEN
       #CycleStart.Started.FillingStarted := FALSE;
       #CycleStart.Started.TemperatureDosingStarted := FALSE;
   END_IF;
   IF #_w4 THEN
       #CycleStart.Started.TransferStarted := FALSE;
       #CycleStart.Started.MIxingStarted := FALSE;
       #CycleStart.Started.RecirculationStarted := FALSE;
   END_IF;
   IF #AlwaysTrue AND #CycleStart.Started.SystemDrainStarted THEN
       #CycleStart.Started.FillingStarted := FALSE;
       #CycleStart.Started.TemperatureDosingStarted := FALSE;
       #CycleStart.Started.TransferStarted := FALSE;
       #CycleStart.Started.MIxingStarted := FALSE;
       #CycleStart.Started.RecirculationStarted := FALSE;
       #CycleStart.Started.DrainStarted := FALSE;
   END_IF;
END_REGION

REGION Network 17: #Over
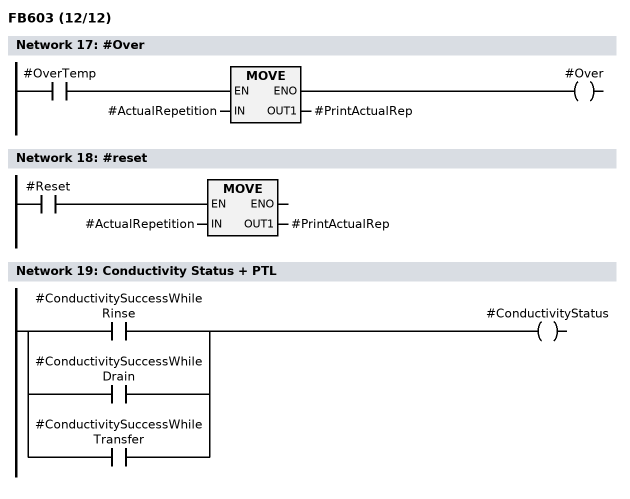
   RUNG wire#powerrail
      Contact( #OverTemp )
      Move(in := #ActualRepetition, out1 => #PrintActualRep)
      Coil( #Over )
   END_RUNG
   // the same network as SCL:
   IF #OverTemp THEN #PrintActualRep := #ActualRepetition; END_IF;
   #Over := #OverTemp;
END_REGION

REGION Network 18: #reset
   RUNG wire#powerrail
      Contact( #Reset )
      Move(in := #ActualRepetition, out1 => #PrintActualRep)
   END_RUNG
   // the same network as SCL:
   IF #Reset THEN #PrintActualRep := #ActualRepetition; END_IF;
END_REGION

REGION Network 19: Conductivity Status + PTL
   RUNG wire#powerrail
      Contact( #ConductivitySuccessWhileRinse )
      wire#w1
      Coil( #ConductivityStatus )
   END_RUNG
   RUNG wire#powerrail
      Contact( #ConductivitySuccessWhileDrain )
   END_RUNG wire#w1
   RUNG wire#powerrail
      Contact( #ConductivitySuccessWhileTransfer )
   END_RUNG wire#w1
   // the same network as SCL:
   #ConductivityStatus := #ConductivitySuccessWhileRinse OR #ConductivitySuccessWhileDrain OR #ConductivitySuccessWhileTransfer;
END_REGION
END_FUNCTION_BLOCK
